		IF NOT Busy 
		THEN (* Busy initalisation is TRUE *)
			Busy := BusyIntern 								:= TRUE;
			state 											:= eSTATE.ABORTING;
		ELSE
			; (* Wait for Startup End*)
		END_IF
	{endregion} 		
	{region "IDLE"} 
	eSTATE.IDLE:
		info 												:= TO_STRING(eSTATE.IDLE);
		
		IF GoToAborting 
		THEN
			Busy := BusyIntern 								:= TRUE; 
			state 											:= eSTATE.ABORTING;
		ELSIF RemoteCtrlEnable AND MasterCmdState = eSTATE.STOPPING 
		THEN
			Busy := BusyIntern 								:= TRUE; 
			state 											:= eSTATE.STOPPING;
		ELSIF NOT RemoteCtrlEnable AND SetMode <> eMODE.IDLE
			OR 
			RemoteCtrlEnable
			AND MasterCmdState <> eSTATE.IDLE
			AND MasterCmdState <> eSTATE.RESETTING
		THEN
			Busy := BusyIntern 								:= TRUE; 
			Mode 											:= SEL(RemoteCtrlEnable,SetMode,MasterCmdMode);
			State 											:= eSTATE.STARTING;
		ELSE
			Mode 											:= eMODE.IDLE;
		END_IF
	{endregion} 
	{region "STARTING"} 	
	eSTATE.STARTING: info 									:= TO_STRING(eSTATE.STARTING);
	
		IF GoToAborting 
		THEN
			state 											:= eSTATE.ABORTING;
			Busy := BusyIntern 								:= TRUE;

		ELSIF RemoteCtrlEnable
			AND(
			MasterCmdState = eSTATE.STOPPING
			OR (* Betriebsartenwechsel ueber RemoteCtrl ein *)
			NOT RemoteDataToSlaves._WORDS[2].8 AND Mode <> MasterCmdMode)
		THEN
			state 											:= eSTATE.STOPPING;
			Busy := BusyIntern 								:= TRUE;
		ELSIF NOT Busy 
		THEN
			state 											:= eSTATE.STARTED;			
		END_IF
	{endregion} 		
	{region "STARTED"} 	
	eSTATE.STARTED: info 									:= TO_STRING(eSTATE.STARTED);
		
		IF GoToAborting 
		THEN
			Busy := BusyIntern 								:= TRUE; 
			state 											:= eSTATE.ABORTING;
		ELSIF RemoteCtrlEnable
			AND NOT RemoteDataToSlaves._WORDS[2].8 
			AND Mode <> MasterCmdMode
		THEN (* Betriebsartenwechsel ueber RemoteCtrl ein *)
			Busy := BusyIntern 								:= TRUE; 
			state 											:= eSTATE.STOPPING;
		ELSIF NOT RemoteCtrlEnable
			OR 	
			RemoteCtrlEnable
			AND MasterCmdState <> eSTATE.STARTED
			AND MasterCmdState <> eSTATE.STARTING
		THEN
			IF RemoteCtrlEnable AND MasterCmdState = eSTATE.EXECUTE
				OR NOT RemoteCtrlEnable
			THEN
				Busy := BusyIntern 							:= TRUE; 
				state 										:= eSTATE.EXECUTE;
			ELSIF RemoteCtrlEnable AND Options.5 //Compl. aktiviert
				AND(MasterCmdState = eSTATE.COMPLETING OR	MasterCmdState = eSTATE.COMPLETE)
			THEN
				Busy := BusyIntern 							:= TRUE; 
				state 										:= eSTATE.COMPLETING;
			ELSE
				Busy := BusyIntern 							:= TRUE; 
				state 										:= eSTATE.STOPPING;
			END_IF
		END_IF
	{endregion} 	
	{region "EXECUTE"} 
	eSTATE.EXECUTE: info 									:= TO_STRING(eSTATE.EXECUTE);
	
		IF GoToAborting 
		THEN
			Busy := BusyIntern 								:= TRUE; 
			state 											:= eSTATE.ABORTING;

		ELSIF SetMode <> Mode
			AND NOT RemoteCtrlEnable
			AND NOT Options.1  (* Modewechsel ueber Stopping/Completing wenn Options.1 nicht gesetzt *)
			OR	
			NOT RemoteCtrlEnable
			AND SetMode = eMODE.IDLE
			OR	
			RemoteCtrlEnable
			AND MasterCmdState <> eSTATE.EXECUTE
			AND MasterCmdState <> eSTATE.STARTING
			AND MasterCmdState <> eSTATE.STARTED
			OR (* Betriebsartenwechsel ueber RemoteCtrl ein *)
			RemoteCtrlEnable
			AND NOT RemoteDataToSlaves._WORDS[2].8 AND Mode <> MasterCmdMode
		THEN
			IF Options.5 (* Mode change over Completing *)
				AND(MasterCmdState = eSTATE.COMPLETING
				AND RemoteCtrlEnable
				OR	
				NOT RemoteCtrlEnable)
			THEN
				Busy := BusyIntern 							:= TRUE; 
				state 										:= eSTATE.COMPLETING;
			ELSE      						
				Busy := BusyIntern 							:= TRUE; 				
				state 										:= eSTATE.STOPPING;
			END_IF

		ELSIF Options.1  (* Modewechsel in Execute *)
			AND(
			SetMode <> Mode AND NOT RemoteCtrlEnable
			OR	
			MasterCmdMode <> Mode AND RemoteCtrlEnable)
		THEN
			Mode 											:= SEL(RemoteCtrlEnable,SetMode,MasterCmdMode);

		ELSIF RemoteCtrlEnable
			AND(
			MasterCmdState = eSTATE.HOLDING 
			OR MasterCmdState = eSTATE.HELD) 
		THEN
			Busy := BusyIntern 								:= TRUE; 
			state 											:= eSTATE.HOLDING;
		ELSIF RemoteCtrlEnable
			AND(
			MasterCmdState = eSTATE.SUSPENDING 
			OR MasterCmdState = eSTATE.SUSPENDED) 
		THEN
			Busy := BusyIntern 								:= TRUE; 
			state 											:= eSTATE.SUSPENDING;
		END_IF
	{endregion} 	
	{region "SUSPENDING"} 
	eSTATE.SUSPENDING: 	info 								:= TO_STRING(eSTATE.SUSPENDING);	
		
		IF GoToAborting 
		THEN
			state 											:= eSTATE.ABORTING;
			Busy := BusyIntern 								:= TRUE;

		ELSIF RemoteCtrlEnable
			AND(
			MasterCmdState = eSTATE.STOPPING
			OR (* Betriebsartenwechsel ueber RemoteCtrl ein *)
			NOT RemoteDataToSlaves._WORDS[2].8 AND Mode <> MasterCmdMode)
		THEN
			state 											:= eSTATE.STOPPING;
			Busy := BusyIntern 								:= TRUE;
		ELSIF NOT Busy 
		THEN
			state 											:= eSTATE.SUSPENDED;		
		END_IF	
	{endregion} 	
	{region "SUSPENDED"} 
	eSTATE.SUSPENDED:	info 								:= TO_STRING(eSTATE.SUSPENDED);	
	
		IF GoToAborting 
		THEN
			Busy := BusyIntern 								:= TRUE; 
			state 											:= eSTATE.ABORTING;
		ELSIF RemoteCtrlEnable
			AND NOT RemoteDataToSlaves._WORDS[2].8 
			AND Mode <> MasterCmdMode
		THEN (* Betriebsartenwechsel ueber RemoteCtrl ein *)
			Busy := BusyIntern 								:= TRUE; 
			state 											:= eSTATE.STOPPING;
		ELSIF NOT RemoteCtrlEnable
			OR 	
			RemoteCtrlEnable
			AND MasterCmdState <> eSTATE.SUSPENDED
			AND MasterCmdState <> eSTATE.SUSPENDING
		THEN
			IF RemoteCtrlEnable 
				AND(MasterCmdState = eSTATE.UNSUSPENDING OR MasterCmdState = eSTATE.EXECUTE OR MasterCmdState = eSTATE.COMPLETING)
				OR NOT RemoteCtrlEnable
			THEN
				Busy := BusyIntern 							:= TRUE; 
				state 										:= eSTATE.UNSUSPENDING;	
			ELSE
				Busy := BusyIntern 							:= TRUE; 
				state 										:= eSTATE.STOPPING;
			END_IF
		END_IF
	{endregion} 	
	{region "UNSUSPENDING"}	
	eSTATE.UNSUSPENDING: info 								:= TO_STRING(eSTATE.UNSUSPENDING);
	
		IF GoToAborting 
		THEN
			state 											:= eSTATE.ABORTING;
			Busy := BusyIntern 								:= TRUE;

		ELSIF RemoteCtrlEnable
			AND(
			MasterCmdState = eSTATE.STOPPING
			OR (* Betriebsartenwechsel ueber RemoteCtrl ein *)
			NOT RemoteDataToSlaves._WORDS[2].8 AND Mode <> MasterCmdMode)
		THEN
			state 											:= eSTATE.STOPPING;
			Busy := BusyIntern 								:= TRUE;
		ELSIF NOT Busy 
		THEN
			Busy := BusyIntern 								:= TRUE; 
			state											:= eSTATE.EXECUTE;
		END_IF
	{endregion} 	
	{region "HOLDING"}	
	eSTATE.HOLDING:		info 								:= TO_STRING(eSTATE.HOLDING);
	
		IF GoToAborting 
		THEN
			state 											:= eSTATE.ABORTING;
			Busy := BusyIntern 								:= TRUE;

		ELSIF RemoteCtrlEnable
			AND(
			MasterCmdState = eSTATE.STOPPING
			OR (* Betriebsartenwechsel ueber RemoteCtrl ein *)
			NOT RemoteDataToSlaves._WORDS[2].8 AND Mode <> MasterCmdMode)
		THEN
			state 											:= eSTATE.STOPPING;
			Busy := BusyIntern 								:= TRUE;
		ELSIF NOT Busy 
		THEN
			state 											:= eSTATE.HELD;		
		END_IF	
	{endregion} 	
	{region "HELD"}	
	eSTATE.HELD:		info 								:= TO_STRING(eSTATE.HELD);
	
		IF GoToAborting 
		THEN
			Busy := BusyIntern 								:= TRUE; 
			state 											:= eSTATE.ABORTING;
		ELSIF RemoteCtrlEnable
			AND NOT RemoteDataToSlaves._WORDS[2].8 
			AND Mode <> MasterCmdMode
		THEN (* Betriebsartenwechsel ueber RemoteCtrl ein *)
			Busy := BusyIntern 								:= TRUE; 
			state 											:= eSTATE.STOPPING;
		ELSIF NOT RemoteCtrlEnable
			OR 	
			RemoteCtrlEnable
			AND MasterCmdState <> eSTATE.HELD
			AND MasterCmdState <> eSTATE.HOLDING
		THEN
			IF RemoteCtrlEnable 
				AND(MasterCmdState = eSTATE.EXECUTE OR MasterCmdState = eSTATE.UNHOLDING OR MasterCmdState = eSTATE.COMPLETING)
				OR NOT RemoteCtrlEnable
			THEN
				Busy := BusyIntern 							:= TRUE; 
				state 										:= eSTATE.UNHOLDING;	
			ELSE
				Busy := BusyIntern 							:= TRUE; 
				state 										:= eSTATE.STOPPING;
			END_IF
		END_IF
	{endregion} 	
	{region "UNHOLDING"}	
	eSTATE.UNHOLDING: 	info 								:= TO_STRING(eSTATE.UNHOLDING);
	
		IF GoToAborting 
		THEN
			state 											:= eSTATE.ABORTING;
			Busy := BusyIntern 								:= TRUE;

		ELSIF RemoteCtrlEnable
			AND(
			MasterCmdState = eSTATE.STOPPING
			OR (* Betriebsartenwechsel ueber RemoteCtrl ein *)
			NOT RemoteDataToSlaves._WORDS[2].8 AND Mode <> MasterCmdMode)
		THEN
			state 											:= eSTATE.STOPPING;
			Busy := BusyIntern 								:= TRUE;
		ELSIF NOT Busy 
		THEN
			Busy := BusyIntern 								:= TRUE; 
			state											:= eSTATE.EXECUTE;
		END_IF
	{endregion} 	
	{region "COMPLETING"}	
	eSTATE.COMPLETING: info 								:= TO_STRING(eSTATE.COMPLETING);
	
		IF GoToAborting 
		THEN
			Busy := BusyIntern 								:= TRUE; 
			state 											:= eSTATE.ABORTING;

		ELSIF RemoteCtrlEnable
			AND( (* Betriebsartenwechsel ueber RemoteCtrl ein *)
			MasterCmdState = eSTATE.STOPPING
			OR 
			NOT RemoteDataToSlaves._WORDS[2].8  AND Mode <> MasterCmdMode)
			OR	
			NOT RemoteCtrlEnable AND NOT Options.5 (* Cancel Completing *)
		THEN
			Busy := BusyIntern 								:= TRUE; 
			state 											:= eSTATE.STOPPING;

		ELSIF NOT Busy
		THEN
			state 											:= eSTATE.COMPLETE;
		END_IF
	{endregion} 	
	{region "COMPLETE"}	
	eSTATE.COMPLETE: info 									:= TO_STRING(eSTATE.COMPLETE);
		
		IF GoToAborting 
		THEN
			Busy := BusyIntern 								:= TRUE; 
			state 											:= eSTATE.ABORTING;

		ELSIF NOT RemoteCtrlEnable
			OR	
			RemoteCtrlEnable
			AND MasterCmdState <> eSTATE.COMPLETE
			AND MasterCmdState <> eSTATE.COMPLETING
		THEN
			Busy := BusyIntern 								:= TRUE; 
			state 											:= eSTATE.STOPPING;
		END_IF
	{endregion} 	
	{region "ABORTING"}	
	eSTATE.ABORTING: info 									:= TO_STRING(eSTATE.ABORTING);
		IF NOT Busy
			OR NOT EStopDelayOK
			OR RemoteCtrlEnable AND NOT MasterCmdInfo.15 (* EStop Delay False *)
		THEN
			StateComplete(); (* Ueber Hardware vorgegeben *)
			state 											:= eSTATE.ABORTED;
		END_IF
			 
		(* Set SubCtrl Busy if state changing *)
		IF state <> eSTATE.ABORTING AND state <> eSTATE.ABORTED 
		THEN 
			Busy := BusyIntern 								:= TRUE; 
		END_IF
			 
	{endregion} 	
	{region "ABORTED"}	
	eSTATE.ABORTED: info 									:= TO_STRING(eSTATE.ABORTED);
		
		IF NOT RemoteCtrlEnable AND EStopDirectOK AND EStopDelayOK
			OR 	
			RemoteCtrlEnable
			AND(EStopDirectOK AND EStopDelayOK OR Options.3)
			AND MasterCmdState <> eSTATE.ABORTED
			AND MasterCmdState <> eSTATE.ABORTING
			AND MasterCmdState <> eSTATE.STARTUP
		THEN
			Busy := BusyIntern 								:= TRUE; 
			state 											:= eSTATE.CLEARING;
		ELSE			
			(* Ack error in aborted *)
			IF LocalReset
			THEN
		 		ErrHdl.reset();
			END_IF
		END_IF
		
		(* set Mode *)
		IF Options.0
		THEN
			Mode 											:= eMODE.IDLE;
		ELSE (* take the current mode back *)
			Mode 											:= SEL(RemoteCtrlEnable,SetMode,MasterCmdMode);
		END_IF
	{endregion} 	
	{region "CLEARING"}	
	eSTATE.CLEARING: info 									:= TO_STRING(eSTATE.CLEARING);
		
		IF GoToAborting 
		THEN
			Busy := BusyIntern 								:= TRUE; 
			state 											:= eSTATE.ABORTING;
		ELSIF NOT Busy
			AND(EStopOK OR Options.3) (* Local EStop Disabled *)
			AND(MasterCmdInfo.14 OR NOT RemoteCtrlEnable) (* RemoteCtrl EStop OK *)
		THEN
			state 											:= eSTATE.STOPPED;
		END_IF
	{endregion} 	
	{region "STOPPING"}	
	eSTATE.STOPPING: Info									:= TO_STRING(eSTATE.STOPPING);
		
		IF GoToAborting 
		THEN
			Busy := BusyIntern 								:= TRUE; 
			state 											:= eSTATE.ABORTING;
		ELSIF NOT Busy 
		THEN
			state 											:= eSTATE.STOPPED;
		END_IF
	{endregion} 	
	{region "STOPPED"}	
	eSTATE.STOPPED: info 									:= TO_STRING(eSTATE.STOPPED);
		
		IF GoToAborting 
		THEN
			Busy := BusyIntern 								:= TRUE; 
			state 											:= eSTATE.ABORTING;
		ELSIF LocalReset AND ErrHdl.flag
			AND(NOT RemoteCtrlEnable OR MasterCmdState <> eSTATE.STOPPED) (* Weiter ueber Quitt im Fehlerfall *)
			AND(ErrHdl.id <> ERROR_MACHINE OR NOT Options.4)
			OR 
			NOT RemoteCtrlEnable
			AND(NOT ErrHdl.flag OR NOT Options.6 AND ErrHdl.id <> ERROR_EXTERNAL) (* Automatisch weiter wenn kein Fehler, oder ACK nicht erforderlich und Fehler nicht Extern (Quittierung erfolgt dort)*)
			OR	
			RemoteCtrlEnable (* Weiter wenn Remote Unit nicht in Stopped/Completing und nicht in Fehler *)
			AND MasterCmdState <> eSTATE.STOPPED
			AND MasterCmdState <> eSTATE.STOPPING
			AND MasterCmdState <> eSTATE.CLEARING
			AND MasterCmdState <> eSTATE.COMPLETING 
			AND MasterCmdState <> eSTATE.COMPLETE
			AND(NOT ErrHdl.flag OR NOT Options.6)
			OR 
			RemoteCtrlEnable (* Weiter wenn Maschinenfehler resetet wird *)
			AND MasterCmdState = eSTATE.RESETTING
			AND ErrHdl.flag //(MasterCmdInfo.11 or MasterCmdInfo.12 OR MasterCmdInfo.13) //OR ErrHdl.id = ERROR_MACHINE ist Bit 12)
		THEN
			Busy := BusyIntern 								:= TRUE; 
			ErrHdl.reset();
			state 											:= eSTATE.RESETTING;
		END_IF
	
		(* set Mode *)
		IF Options.0 
		THEN
			Mode 											:= eMODE.IDLE;
		ELSE (* take the current mode back *)
			Mode 											:= SEL(RemoteCtrlEnable,SetMode,MasterCmdMode);
		END_IF
	{endregion} 	
	{region "RESETTING"}	
	eSTATE.RESETTING: info 									:= TO_STRING(eSTATE.RESETTING);
		
		IF GoToAborting 
		THEN
			Busy := BusyIntern 								:= TRUE; 
			state 											:= eSTATE.ABORTING;
		ELSIF MasterCmdState = eSTATE.STOPPING 
			AND RemoteCtrlEnable 
		THEN
			Busy := BusyIntern 								:= TRUE; 
			state 											:= eSTATE.STOPPING;
		ELSIF NOT Busy 
		THEN
			state 											:= eSTATE.IDLE;
		END_IF
	{endregion} 	

	ELSE
		info 												:= CONCAT('ERROR unkown state ', TO_STRING(state));
		ErrHdl.flag 										:= TRUE;
		ErrHdl.fnc 											:= 'SubCtrl';
		ErrHdl.id											:= 99;
		ErrHdl.state										:= state;
		ErrHdl.text 										:= CONCAT('unkown state:',DINT_TO_STRING(ErrHdl.state));
		SetLocalError();
	END_CASE
		 
(* State Check *************************************************)
	RT_StateChanged 										:= LastState <> State;
	LastState 												:= State;
	
(* Statebits ***********************************************************************************)
	InStartup												:= state = eSTATE.STARTUP;
	InIdle													:= state = eSTATE.IDLE;
	InStarting												:= state = eSTATE.STARTING;
	InStarted												:= state = eSTATE.STARTED;
	InExecute												:= state = eSTATE.EXECUTE;
	InCompleting											:= state = eSTATE.COMPLETING;
	InComplete												:= state = eSTATE.COMPLETE;
	InAborting												:= state = eSTATE.ABORTING;
	InAborted												:= state = eSTATE.ABORTED;
	InClearing												:= state = eSTATE.CLEARING;
	InStopping												:= state = eSTATE.STOPPING;
	InStopped												:= state = eSTATE.STOPPED;
	InResetting												:= state = eSTATE.RESETTING;

	EStopStartupOK											:= 	NOT InAborted 
																AND(
																EStopStartupOK 
																OR 
																NOT InAborting AND NOT InClearing 
																AND NOT InStartup AND NOT InStopped );
                    										
(* optional
	InSuspending	:= state = eSTATE.SUSPENDING;
	InSuspended		:= state = eSTATE.SUSPENDED;
	InUnsuspending	:= state = eSTATE.UNSUSPENDING;

	InHolding		:= state = eSTATE.HOLDING;
	InHeld			:= state = eSTATE.HELD;
	InUnholding		:= state = eSTATE.UNHOLDING;
*)

(***************************************************************)
(* Read Subs Status and synchronize							   *)
(***************************************************************)		
{region "Check slave states and send command"}	
	(* Init Flag, all Subs in same state *)
	NoSlavesConnected										:= TRUE;
	SlavesInSync 											:= NOT RT_StateChanged;
	SlavesBusy    											:= FALSE;
	NoOfBusySlaves											:= 0;
	(* Init remote command data to slaves  *)
	RemoteDataToSlaves._INTs[0]								:= Mode;
	RemoteDataToSlaves._WORDS[2]							:= TO_WORD(Options);
	RemoteDataToSlaves._WORDS[2].8							:= RemoteCtrlEnable;
	RemoteDataToSlaves._WORDS[2].9							:= LocalReset;	
	RemoteDataToSlaves._WORDS[2].14							:= EStopOK OR Options.3;
	RemoteDataToSlaves._WORDS[2].15							:= EStopDelayOK OR Options.3;	
	RemoteDataToSlaves._INTs[3]								:= Id;
		
	(* read Subs state an send cmd to all subs *)
	FOR i := MIN_SLAVE TO MAX_SLAVE DO
		IF ipSlave[i] <> 0 
		THEN 
			NoSlavesConnected 								:= FALSE;(* pointer is used *)
			RemoteDataFromSlave								:= ipSlave[i].remoteData; //Read remote status data from slaves
			IF RemoteDataFromSlave._WORDS[2].8 
			THEN (* External Sub is Remote-Controlled *)
				(* Check the status from then external subs *)
				IF((RemoteDataFromSlave._WORDS[2].11 OR RemoteDataFromSlave._WORDS[2].13) 
					AND RemoteDataFromSlave._WORDS[2].4)(* Maschine to Remotesystem if Enabled, or External Error *)
					AND NOT ErrHdl.flag
					AND NOT InStartup AND NOT InResetting
					AND NOT InAborting AND NOT InAborted
				THEN (* external sub has fatal error *)
					(* external subs send fatal machine error -> bring local sub in Stopping with error *)
					ErrHdl.flag								:= TRUE;
					ErrHdl.state							:= state;
					ErrHdl.fnc 								:= name;
					ErrHdl.id								:= ERROR_EXTERNAL;
					ErrHdl.text 							:= CONCAT('Fatal machine error in Sub index no.:',INT_TO_STRING(i));
					Busy									:= state <> eSTATE.STOPPING;
					state 									:= eSTATE.STOPPING;
					SlavesInSync 							:= FALSE;
				ELSE (* external sub has no error *)
					IF SlavesState = RemoteDataFromSlave._INTs[1]
					THEN (* Check if sub is in sync with other subs *)
						SlavesState 						:= RemoteDataFromSlave._INTs[1];
					ELSE (* external sub is not in sync with other subs *)
						IF (RemoteDataFromSlave._INTs[1] = eSTATE.ABORTED OR RemoteDataFromSlave._INTs[1] = eSTATE.ABORTING)
							AND NOT InAborted 
							AND NOT InAborting
							AND NOT RemoteDataFromSlave._WORDS[2].3 (* Local EStop-Signals Disable *)
							OR RemoteDataFromSlave._WORDS[2].11 (* Maschine Error *)
							OR RemoteDataFromSlave._WORDS[2].12 (* Local Error  *)
							OR RemoteDataFromSlave._WORDS[2].13 (* External Error  *)
							OR (* comleting at sub disabled *)
							NOT RemoteDataFromSlave._WORDS[2].5 
							AND(InCompleting OR InComplete)
							AND(RemoteDataFromSlave._INTs[1] = eSTATE.STOPPING OR RemoteDataFromSlave._INTs[1] = eSTATE.STOPPED)
						THEN
							; (* ignore cause sub use local EStop-signals, or error in stopped *)
						ELSE
							SlavesState						:= RemoteDataFromSlave._INTs[1];
							SlavesInSync 					:= FALSE;
						END_IF
					END_IF

					(* subs busy *)
					IF (RemoteDataFromSlave._INTs[1] = eSTATE.ABORTED OR RemoteDataFromSlave._INTs[1] = eSTATE.ABORTING )
						AND NOT InAborted 
						AND NOT InAborting
						AND NOT RemoteDataFromSlave._WORDS[2].3 (* Local EStop-Signals Disable *)
						OR RemoteDataFromSlave._WORDS[2].12 (* Local Error *)
						OR 
						SlavesState = eSTATE.EXECUTE AND NOT InExecute
					THEN
						; (* ignore cause sub is in error or use local EStop-Signals *)
					ELSIF RemoteDataFromSlave._WORDS[2].10 
					THEN
						SlavesBusy 							:= TRUE;
						NoOfBusySlaves						:= NoOfBusySlaves + 1;
					END_IF

				END_IF
			ELSE (* external Sub is not in RemoteCtrl *)
				;
			END_IF

			(* Write latest command data   *)
			RemoteDataToSlaves._INTs[1]						:= State;
			RemoteDataToSlaves._WORDS[2].10					:= Busy;
			RemoteDataToSlaves._WORDS[2].11					:= ErrHdl.id = ERROR_MACHINE;
			RemoteDataToSlaves._WORDS[2].12					:= ErrHdl.id = ERROR_LOCAL;
			RemoteDataToSlaves._WORDS[2].13					:= ErrHdl.id = ERROR_EXTERNAL;

			(* set slave command data *)
			ipSlave[i].remoteData							:= RemoteDataToSlaves; //Write data as command to every slave
		ELSE
			EXIT; (* pointer not used -> Exit for *)
		END_IF
	END_FOR

	(* Set state complete only if all Subs in the same state or current state is Execute *)
	IF SlavesInSync AND NOT NoSlavesConnected 
	THEN //Subs in sync
		IF SlavesBusy 
			OR (BusyIntern AND Options.2) 
			OR (NOT EStopOK AND NOT Options.3 AND InClearing) (* Solange Busy halten, biss durch EStopOK aus Clearing gegangen werden kann *)
		THEN
			; (* al least one sub is busy or not StateComplete *)
		ELSIF Busy 
		THEN
			Busy := BusyIntern 								:= FALSE; (* All subs not StateComplete (NOT Busy) set UnitSub StateComplete *)
		END_IF
	END_IF
{endregion}
	 
(* Set Status RemoteData for master to check ************************************************************)
	RemoteDataToSlaves._INTs[0] 							:= Mode;
	RemoteDataToSlaves._INTs[1]								:= State;
	RemoteDataToSlaves._WORDs[2]							:= TO_WORD(Options);
	RemoteDataToSlaves._WORDs[2].8							:= RemoteCtrlEnable;
	RemoteDataToSlaves._WORDs[2].9							:= LocalReset;
	RemoteDataToSlaves._WORDs[2].10							:= Busy;
	RemoteDataToSlaves._WORDs[2].11							:= ErrHdl.id = ERROR_MACHINE;
	RemoteDataToSlaves._WORDs[2].12							:= ErrHdl.id = ERROR_LOCAL;
	RemoteDataToSlaves._WORDs[2].13							:= ErrHdl.id = ERROR_EXTERNAL;
	RemoteDataToSlaves._WORDs[2].14							:= EStopOK OR Options.3;
	RemoteDataToSlaves._WORDs[2].15							:= EStopDelayOK OR Options.3;
	RemoteDataToSlaves._INTs[3]								:= Id;
	

(* Reset LocalAck ******************************************************************************)
	Localreset												:= FALSE;

(***********************************************************************************************)

METHOD PRIVATE FINAL _createID : INT
VAR_STAT //Value is stored for each instance
	IdCnt													: INT;
END_VAR
IdCnt														:= IdCnt + 1;
_CreateID 													:= IdCnt;
END_METHOD

METHOD PUBLIC FINAL addSlave : BOOL
VAR_INPUT
	ipSlave													:	I_Statemodel;
END_VAR
addSlave													:= FALSE;	
IF ipSlave <> 0	
then
	FOR i := MIN_SLAVE TO MAX_SLAVE
	DO 
		IF ipSlave = THIS^.ipSlave[i] THEN
			addSlave										:= TRUE;
			EXIT;
		ELSIF THIS^.ipSlave[i] = 0
		THEN								
			THIS^.ipSlave[i]								:= ipSlave;
			addSlave										:= TRUE;
			EXIT;
		END_IF
	END_FOR
END_IF
END_METHOD

METHOD FB_init : BOOL
VAR_INPUT
	bInitRetains : BOOL; // if TRUE, the retain variables are initialized (warm start / cold start)
	bInCopyCode : BOOL;  // if TRUE, the instance afterwards gets moved into the copy code (online change)
END_VAR
(* Generate ID ****************************************************)
	IF Id = 0 
	THEN 
		id 													:= _CreateID(); 
		IF Name = '' 
		THEN 
			Name 											:= CONCAT('Statemodel Id ',TO_STRING(Id)); 
		ELSE
			Name 											:= CONCAT(Name , CONCAT(' Id ', TO_STRING(Id))); 
		END_IF
	END_IF	
(***********************************************************************)
END_METHOD

METHOD PUBLIC goToStopping : BOOL //TRUE = stopping activated
VAR_INPUT
END_VAR

CASE State OF
eSTATE.IDLE,
eSTATE.STARTING,
eSTATE.STARTED,	
eSTATE.EXECUTE,
eSTATE.SUSPENDING,
eSTATE.SUSPENDED,
eSTATE.UNSUSPENDING,	
eSTATE.HOLDING,
eSTATE.HELD,
eSTATE.UNHOLDING,	
eSTATE.COMPLETING,
eSTATE.COMPLETE,
eSTATE.STOPPING,
eSTATE.STOPPED,
eSTATE.RESETTING:
	state 													:= eSTATE.STOPPING;
	Busy := BusyIntern 										:= TRUE;
	goToStopping											:= TRUE;
ELSE
(*	
	eSTATE.STARTUP,
	eSTATE.ABORTING,
	eSTATE.ABORTED,
	eSTATE.CLEARING:
*)	
	goToStopping											:= FALSE;
END_CASE
END_METHOD

METHOD PUBLIC isModeActive : BOOL
VAR_INPUT
	Mode													: eMODE;				
END_VAR
IsModeActive := Mode = THIS^.Mode AND(InExecute OR InCompleting);
END_METHOD

METHOD PUBLIC isStateActive : BOOL
VAR_INPUT
	state								: eSTATE;
END_VAR
IsStateActive := state = This^.State;
END_METHOD

METHOD PUBLIC reset : boOL //Result = TRUE if Resetting finished - ErrHdl.Flag = FALSE
VAR_INPUT
END_VAR
LocalReset													:= TRUE;
reset														:= NOT ErrHdl.flag;
END_METHOD

METHOD PUBLIC setLocalError : booL
VAR_INPUT
END_VAR
IF NOT ErrHdl.flag
	AND state <> eSTATE.ABORTING
	AND state <> eSTATE.ABORTED
	AND state <> eSTATE.CLEARING
	and state <> eSTATE.RESETTING
THEN
	ErrHdl.flag 											:= TRUE;
	ErrHdl.state											:= state;
	ErrHdl.fnc												:= name;
	ErrHdl.id												:= ERROR_LOCAL;
	ErrHdl.text 											:= 'Local ctrl error';
	Busy													:= state <> eSTATE.STOPPING;
	state 													:= eSTATE.STOPPING;
	SetLocalError											:= TRUE;
ELSE
	SetLocalError											:= ErrHdl.id = ERROR_LOCAL;
END_IF
END_METHOD

METHOD PUBLIC setMachineError : booL
VAR_INPUT
END_VAR
IF NOT ErrHdl.flag
	AND state <> eSTATE.ABORTING
	AND state <> eSTATE.ABORTED
	AND state <> eSTATE.CLEARING
	AND state <> eSTATE.RESETTING
THEN
	ErrHdl.flag												:= TRUE;
	ErrHdl.state											:= state;
	ErrHdl.fnc												:= name;
	ErrHdl.id												:= ERROR_MACHINE;
	ErrHdl.text 											:= 'Fatal machine error';
	Busy													:= state <> eSTATE.STOPPING;
	state 													:= eSTATE.STOPPING;
	SetMachineError											:= TRUE;
ELSE
	SetMachineError											:= ErrHdl.id = ERROR_MACHINE;;
END_IF
END_METHOD

METHOD PUBLIC FINAL stateComplete : BOOL //Result = TRUE if state completed (BusyIntern=FALSE)
VAR_INPUT
END_VAR
BusyIntern 													:= FALSE;
StateComplete												:= NOT BusyIntern AND NOT Busy;
END_METHOD

{attribute 'monitoring' := 'call'}
PROPERTY PUBLIC optDisableSafetyInputs : BOOL
GET
optDisableSafetyInputs := Options.3;
END_GET
SET
Options.3 := optDisableSafetyInputs;
END_SET
END_PROPERTY

{attribute 'monitoring' := 'call'}
PROPERTY PUBLIC optEnableAutoChangeModeToIdle : BOOL
GET
optEnableAutoChangeModeToIdle := Options.0;
END_GET
SET
Options.0 := optEnableAutoChangeModeToIdle;
END_SET
END_PROPERTY

{attribute 'monitoring' := 'call'}
PROPERTY PUBLIC optEnableExplicitReset : BOOL
GET
optEnableExplicitReset := Options.6;
END_GET
SET
Options.6 := optEnableExplicitReset;
END_SET
END_PROPERTY

{attribute 'monitoring' := 'call'}
PROPERTY PUBLIC optEnableExternalStateComplete : BOOL
GET
optEnableExternalStateComplete := Options.2;
END_GET
SET
Options.2 := optEnableExternalStateComplete;
END_SET
END_PROPERTY

{attribute 'monitoring' := 'call'}
PROPERTY PUBLIC optEnableFwdMachineErrorToMaster : BOOL
GET
optEnableFwdMachineErrorToMaster := Options.4;
END_GET
SET
Options.4 := optEnableFwdMachineErrorToMaster;
END_SET
END_PROPERTY

{attribute 'monitoring' := 'call'}
PROPERTY PUBLIC optEnableModeChangeInExecute : BOOL
GET
optEnableModeChangeInExecute := Options.1;
END_GET
SET
Options.1 := optEnableModeChangeInExecute;
END_SET
END_PROPERTY

{attribute 'monitoring' := 'call'}
PROPERTY PUBLIC optEnableModeChangeViaStateCompl : BOOL
GET
optEnableModeChangeViaStateCompl := Options.5;
END_GET
SET
Options.5 := optEnableModeChangeViaStateCompl;
END_SET
END_PROPERTY

{attribute 'monitoring' := 'call'}
PROPERTY PUBLIC optEnableSetActState : BOOL
GET
optEnableSetActState := Options.7;
END_GET
SET
Options.7 := optEnableSetActState;
END_SET
END_PROPERTY

{attribute 'monitoring' := 'call'}
PROPERTY public actMode : eMODE
GET
actMode := Mode;
END_GET
END_PROPERTY

{attribute 'monitoring' := 'call'}
//Actual state enum, only read access by default, check options for further information 
PROPERTY public actState : eSTATE
GET
actState := state;
END_GET
SET
PUBLIC //Use with care!! 
VAR
END_VAR
IF Options.7  //OPTION_ENABLE_SET_ACT_STATE
THEN
	IF actState <> State
	THEN
		state 													:= actState;
		Busy := BusyIntern 										:= TRUE;	
	END_IF
ELSE	
	ErrHdl.flag 												:= TRUE;
	ErrHdl.state												:= state;
	ErrHdl.fnc													:= name;
	ErrHdl.id													:= ERROR_LOCAL;
	ErrHdl.text 												:= 'Write "actState" not allowed, use OPTION_ENABLE_SET_ACT_STATE to enable set actState';
	Busy														:= state <> eSTATE.STOPPING;
	state 														:= eSTATE.STOPPING;
END_IF
END_SET
END_PROPERTY

{attribute 'monitoring' := 'call'}
PROPERTY PUBLIC ipMasterUnit : I_Statemodel //The slave will add his interface pointer into the master through this propertiy
SET
IF IdRemoteMaster = 0 AND_THEN ipMasterUnit <> 0
THEN
	RemoteDataToSlaves									:= ipMasterUnit.remoteData;	
	IF IdRemoteMaster <> RemoteDataToSlaves._INTs[3] 
	THEN
		IF ipMasterUnit.addSlave(THIS^)
		THEN					
			remoteData 									:= RemoteDataToSlaves; 
		END_IF
	END_IF
END_IF
END_SET
END_PROPERTY

{attribute 'monitoring' := 'call'}
PROPERTY isBusy : BOOL
GET
isBusy := Busy;
END_GET
END_PROPERTY

PROPERTY public remoteData : U_64BIT_DATATYPE
GET
//statis of sub
remoteData := RemoteDataToSlaves;
END_GET
SET
//Cmd to sub
MasterCmdMode 	:= remoteData._INTs[0];
MasterCmdState := remoteData._INTs[1];
MasterCmdInfo 	:= remoteData._WORDS[2];
IdRemoteMaster := remoteData._INts[3];
END_SET
END_PROPERTY

{attribute 'monitoring' := 'call'}
PROPERTY PUBLIC rErrHdl : REFERENCE to ERROR_HDL
GET
rErrHdl REF= Errhdl;
END_GET
END_PROPERTY

PROPERTY PUBLIC setStateComplete : BOOL
GET
SetStateComplete := not BusyIntern and not Busy;
END_GET
SET
IF SetStateComplete AND BusyIntern
THEN
	StateComplete();
END_IF
END_SET
END_PROPERTY

END_FUNCTION_BLOCK

// POUs/Statemodel/control/I_Statemodel
INTERFACE I_Statemodel extends I_StatemodelBase

METHOD PUBLIC FINAL addSlave : BOOL
VAR_INPUT
	ipSlave					:	I_Statemodel;
END_VAR
END_METHOD

METHOD PUBLIC isModeActive : BOOL
VAR_INPUT
	Mode													: eMODE;				
END_VAR
END_METHOD

METHOD PUBLIC isStateActive : BOOL
VAR_INPUT
	state						:	eSTATE;
END_VAR
END_METHOD

METHOD PUBLIC reset : boOL //Result = TRUE if Resetting finished - ErrHdl.Flag = FALSE
VAR_INPUT
END_VAR
END_METHOD

METHOD PUBLIC setLocalError : booL
VAR_INPUT
END_VAR
END_METHOD

PROPERTY public remoteData : U_64BIT_DATATYPE
GET
END_GET
SET
END_SET
END_PROPERTY

{attribute 'monitoring' := 'call'}
PROPERTY PUBLIC rErrHdl : REFERENCE to ERROR_HDL
GET
END_GET
END_PROPERTY

END_INTERFACE

// POUs/Statemodel/control/I_StatemodelBase
INTERFACE I_StatemodelBase Extends __System.IQueryInterface

METHOD PUBLIC setMachineError : booL
VAR_INPUT
END_VAR
END_METHOD

METHOD PUBLIC stateComplete : BOOL //Result = TRUE if state completed (BusyIntern=TRUE)
VAR_INPUT
END_VAR
END_METHOD

{attribute 'monitoring' := 'call'}
PROPERTY public actMode : eMODE
GET
END_GET
END_PROPERTY

{attribute 'monitoring' := 'call'}
//Actual state enum, only read access by default, check options for further options 
PROPERTY public actState : eSTATE
GET
END_GET
SET
END_SET
END_PROPERTY

{attribute 'monitoring' := 'call'}
PROPERTY isBusy : BOOL
GET
END_GET
END_PROPERTY

PROPERTY PUBLIC setStateComplete : BOOL
GET
END_GET
SET
END_SET
END_PROPERTY

END_INTERFACE

// POUs/Statemodel/UnitTemplate/Statemodel_Unit
{attribute 'no_check'}
//Generic Unit 
FUNCTION_BLOCK Statemodel_Unit implements I_Statemodel_Unit
VAR_OUTPUT CONSTANT
END_VAR             										
VAR_INPUT           										
	unit																:	Statemodel;		
END_VAR             										
VAR_OUTPUT          										
END_VAR             	
VAR                 	
(* Local variables ************************************************************)

(* Trigger *****************************************************************)

(* Timer ******************************************************************)

(* Fcuntion blocks ***************************************************************)

(* Dummys **********************************************************)

END_VAR

	(* Generic unit incl. state model										V1.0		*)
	(************************************************************************************)

(* work local sub ****************************************)
	Unit();
	IF Unit.RT_StateChanged THEN stateChanged(unit.Mode, Unit.State); END_IF
	
(* call methods ********************************************)
	CASE Unit.state OF
	eSTATE.STARTUP			:	Startup();
	eSTATE.IDLE				: 	Idle();
	eSTATE.STARTING			:	Starting();		
	eSTATE.STARTED			: 	Started();	
	eSTATE.EXECUTE			:	Executing();
	eSTATE.COMPLETING		:	Completing();
	eSTATE.COMPLETE			: 	Complete();
	eSTATE.ABORTING			:	Aborting();
	eSTATE.ABORTED			:  	Aborted();
	eSTATE.CLEARING			:	Clearing();
	eSTATE.STOPPING			:	Stopping();
	eSTATE.STOPPED			: 	Stopped();
	eSTATE.RESETTING		:	Resetting();
	ELSE
		;
	END_CASE

(*********************************************************)

METHOD PROTECTED aborted : BOOL
VAR_INPUT
END_VAR
Aborted														:= unit.InAborted;
END_METHOD

METHOD PROTECTED aborting : BOOL
VAR_INPUT
END_VAR
Unit.StateComplete();
Aborting													:= Unit.InAborting;
END_METHOD

METHOD PROTECTED clearing : Bool
VAR_INPUT
END_VAR
Unit.StateComplete();
Clearing													:= Unit.InClearing;
END_METHOD

METHOD PROTECTED complete : Bool
VAR_INPUT
END_VAR
Complete														:= unit.InComplete;
END_METHOD

METHOD PROTECTED completing : BOOL
VAR_INPUT
END_VAR
Unit.StateComplete();
Completing													:= Unit.InCompleting;
END_METHOD

METHOD PROTECTED executing : booL
VAR_INPUT
END_VAR
Executing 												:= Unit.InExecute;
END_METHOD

METHOD FB_exit : BOOL
VAR_INPUT
	bInCopyCode : BOOL; // if TRUE, the exit method is called for exiting an instance that is copied afterwards (online change).
END_VAR
FB_EXit															:= TRUE;
END_METHOD

METHOD FB_init : BOOL
VAR_INPUT
	bInitRetains : BOOL; // if TRUE, the retain variables are initialized (warm start / cold start)
	bInCopyCode : BOOL;  // if TRUE, the instance afterwards gets moved into the copy code (online change)
END_VAR
(* Example 
	Unit.pSubRemoteData[1]												:= ADR(Infeed.unit.RemoteData);
	Unit.pSubRemoteData[2]												:= ADR(Support_1.unit.RemoteData);
	Unit.pSubRemoteData[3]												:= ADR(Support_2.RemoteData);	
	Unit.pSubRemoteData[4]												:= ADR(Transport.unit.RemoteData);
	Unit.pSubRemoteData[5]												:= ADR(Outfeed.unit.RemoteData);
*)
FB_init														:= TRUE;
END_METHOD

METHOD FB_reinit : BOOL
VAR_INPUT
END_VAR
FB_reinit											:= TRUE;
END_METHOD

METHOD PROTECTED idle : Bool
VAR_INPUT
END_VAR
Idle														:= unit.InIdle;
END_METHOD

METHOD PROTECTED Resetting : Bool
VAR_INPUT
END_VAR
Unit.StateComplete();
Resetting													:= Unit.InResetting;
END_METHOD

{attribute 'monitoring' := 'call'}
PROPERTY public rUnit : REFERENCE TO Statemodel
GET
rUnit REF= Unit;
END_GET
END_PROPERTY

METHOD PROTECTED started : Bool
VAR_INPUT
END_VAR
Started													:= Unit.InStarted;
END_METHOD

METHOD PROTECTED starting : Bool
VAR_INPUT
END_VAR
Unit.StateComplete();
Starting													:= Unit.InStarting;
END_METHOD

METHOD PROTECTED startup : Bool
VAR_INPUT
END_VAR
Unit.StateComplete();
Startup													:= Unit.InStartup;
END_METHOD

METHOD PROTECTED stateChanged : BOOL 
VAR_INPUT
	mode											:	eMODE;
	state											:	eSTATE;
END_VAR
END_METHOD

METHOD PROTECTED stopped : Bool
VAR_INPUT
END_VAR
Stopped														:= unit.InStopped;
END_METHOD

METHOD PROTECTED stopping : Bool
VAR_INPUT
END_VAR
Unit.StateComplete();
Stopping													:= Unit.InStopping;
END_METHOD

END_FUNCTION_BLOCK

// POUs/Statemodel/UnitTemplate/I_Statemodel_Unit
INTERFACE I_Statemodel_Unit Extends __System.IQueryInterface

{attribute 'monitoring' := 'call'}
PROPERTY public rUnit : REFERENCE TO Statemodel
GET
END_GET
END_PROPERTY

END_INTERFACE

// POUs/Motion/TF50xx-NC/03_Utilities/CoordinateTransformation2D
FUNCTION_BLOCK CoordinateTransformation2D //CoordinateTransformation
// transformation of an X/Y product coordinate to the machine coordinate system
// MCS = machine coordinate system
// PCS = product coordinate system
VAR_INPUT
//Parameter
	x0 														: LREAL;		// origin MCS X coordinate of the product coordinate system
	y0 														: LREAL;		// origin MCS Y coordinate of the product coordinate system
	x1 														: LREAL;		// opposite corner point MCS X coordinate of the product 
	y1 														: LREAL;		// opposite corner point MCS Y coordinate of the product
	a 														: LREAL;		// length of the product (difference x1pcs-x0pcs)
	b 														: LREAL;		// width of the product (difference y1pcs-y0pcs)
END_VAR                                                 	
VAR_OUTPUT                                              	
	Xmcs 													: LREAL;	// X coordinate in machine coordinate system
	Ymcs 													: LREAL;	// Y coordinate in machine coordinate system
															
	Xpcs 													: LREAL;	// X coordinate in Product coordinate system
	Ypcs 													: LREAL;	// Y coordinate in Product coordinate system
                                                        	
	Alfa													: LREAL;	

	Error 													: BOOL;	
//		ErrorID 											: UDINT;
END_VAR
VAR
	c														: LREAL;
	diagonal												: LREAL;

	ratio													: LREAL;
	
	alfa1													: LREAL;
	alfa2													: LREAL;
END_VAR

;

{attribute 'monitoring' := 'call'}
PROPERTY PUBLIC diagonalMSC : LREAL
GET
VAR
	t		:	LREAL;
END_VAR
t 			:=  EXPT(X1-X0,2.0) + EXPT(y1-y0,2.0);
DiagonalMSC := SQRT(t);
END_GET
END_PROPERTY

{attribute 'monitoring' := 'call'}
PROPERTY PUBLIC diagonalPCS : LREAL
GET
DiagonalPCS := SQRT((a*a)+(b*b));
END_GET
END_PROPERTY

{attribute 'monitoring' := 'call'}
PROPERTY PUBLIC isParamValid : BOOL
GET
IsParamValid 													:= not ParamHasError;
END_GET
SET
PUBLIC 
VAR
END_VAR
IF NOT IsParamValid
THEN
	a 														:= 0.0;
	b 														:= 0.0;
	x1 														:= Y1 := 0.0;
	y0 														:= X0 := 0.0;
END_IF
END_SET
END_PROPERTY

METHOD MSCtoPCS : BOOL //Return value = TRUE if execution finished successful / FALSE if finished with error
VAR_INPUT
	Xmcs 													: LREAL;	// X coordinate in machine coordinate system
	Ymcs 													: LREAL;	// Y coordinate in machine coordinate system
END_VAR
IF ParamHasError THEN
	Error 													:= TRUE; 
	MSCtoPCS 												:= FALSE;
ELSE	
	THIS^.Xmcs												:= Xmcs;	
	THIS^.Ymcs												:= Ymcs;	

	c 														:= SQRT(a*a + b*b);
	alfa 													:= ACOS((x1-x0) / c) - ACOS( a / c);
	
	Xpcs 													:= 	 (Xmcs - x0) * COS(alfa) + (Ymcs - y0) * SIN(alfa);
	Ypcs 													:= - (Xmcs - x0) * SIN(alfa) + (Ymcs - y0) * COS(alfa);
	
	Error 													:= FALSE; 
	MSCtoPCS 												:= TRUE;
END_IF
END_METHOD

{attribute 'monitoring' := 'call'}
PROPERTY PRIVATE paramHasError : BOOL
GET
ParamHasError := 	a<=0.0 
			OR 	b<=0.0 
			OR 	x1=x0 
			OR 	y1=y0;
END_GET
END_PROPERTY

METHOD PUBLIC PCStoMSC : booL //Return value = TRUE if execution finished successful / FALSE if finished with error
VAR_INPUT
	Xpcs : LREAL;	// X coordinate in product coordinate system
	Ypcs : LREAL;	// Y coordinate in product coordinate system	
END_VAR
IF ParamHasError 
THEN
	Error 													:= TRUE; 
	PCStoMSC												:= FALSE;
ELSE                										
	THIS^.Xpcs												:= Xpcs;	
	THIS^.Ypcs												:= Ypcs;
	
	c 														:= SQRT(a*a + b*b);
	diagonal												:= SQRT((x1-x0)*(x1-x0)+(y1-y0)*(y1-y0));
	
	ratio													:= diagonal/c;
	
	alfa1 													:= ACOS((x1-x0) / diagonal);
	alfa2													:= ACOS(a/c);
	
	alfa													:= alfa1-alfa2;
	
	Xmcs 													:= x0 + ratio * (Xpcs * COS(alfa) - Ypcs * SIN(alfa));
	Ymcs 													:= y0 + ratio * (Xpcs * SIN(alfa) + Ypcs * COS(alfa));
                    	
	Error 													:= FALSE; 
	PCStoMSC												:= TRUE;
END_IF
END_METHOD

END_FUNCTION_BLOCK

// POUs/Motion/TF50xx-NC/03_Utilities/getOvrVelo
{attribute 'no_check'}
//Overwrite function - Returns velocity setpoint based on max velo and requested overwrite 
FUNCTION getOvrVelo : LREAL
VAR_INPUT
	SetVelo													:	LREAL;
	MaxVelo													:	LREAL;
END_VAR
VAR
END_VAR

IF 	MaxVelo = 0.0 OR SetVelo = 0.0
THEN
	GetOvrVelo 												:= 0.0;
ELSE                										
	GetOvrVelo 												:= 100.0 / MaxVelo * SetVelo;
END_IF

END_FUNCTION

// POUs/Motion/TF50xx-NC/AxNcBase
FUNCTION_BLOCK AxNcBase EXTENDS AXIS_REF IMPLEMENTS I_AxNcBase(* See Tc2_MC2 *)
VAR_OUTPUT CONSTANT
	OPTION_EN_CMD_ABORTED_ERROR								: 	BYTE := 2#1000_0000; //Default: .7 = xxx.CmdAborted is treaded as error
END_VAR
VAR_INPUT
{attribute 'displaymode':='binary'}
	Options													: 	BYTE  := OPTION_EN_CMD_ABORTED_ERROR; //See output constant for Options mask
	
(* Axis *)
	Admin													: 	AxAdmin;
	para													: 	AxPara;

	Home													:	AxHoming;
	event													:	AxEventHandling;                                                   
END_VAR                                             	
VAR_OUTPUT                                          	
	ErrHdl													:	ERROR_HDL;
END_VAR
VAR
END_VAR

	(* Axis 																*)
	(************************************************************************)

	
(********************************************************************************)
(* Error NC																		*)
(********************************************************************************)
	Event(
		Enable		:= Admin.EnableOK OR Event.NoOfActiveEvents > 0,
		ConfirmTrig	:= Admin.ResetTrig,
		Name		:= para.Name,
		SourceId	:= (* Default *) ,
		rAxis		:= THIS^,
		ErrorId		:= TO_UDINT(ErrHdl.Id),
		Status		=> );
		
	(* Init ErrHdl *)
	ErrHdl.Reset();

(********************************************************************************)
(* work Admin ctrl 																*)
(********************************************************************************)
	Admin(rAxis		:= THIS^);
	IF Admin.Error
	THEN
		ErrHdl.id 											:= UDINT_TO_DINT(Admin.ErrorId);
		ErrHdl.fnc											:= 'Admin';
		ErrHdl.text											:= Admin.ErrorText;
		ErrHdl.flag											:= TRUE;
	END_IF
	
(********************************************************************************)
(* Parameter																	*)
(********************************************************************************)
	para(Axisid := NcToPlc.AxisId);
		
(********************************************************************************)
(* work homing ctrl 															*)
(********************************************************************************)
	Home(rAxis := THIS^ );
	errorCheck(AxBase := Home);
	

(********************************************************************************)

METHOD PROTECTED errorCheck : BOOL
VAR_IN_OUT
	AxBase									:	AxFbBase;
END_VAR
IF AxBase.Error
THEN
	ErrHdl.flag									:= TRUE;
	ErrHdl.fnc									:= 'AxNcPtP';
	ErrHdl.id									:= TO_DINT(AxBase.ErrorID);
	ErrHdl.text									:= AxBase.ErrorText;
	errorCheck									:= TRUE;
ELSIF AxBase.CmdAborted AND Options.7
THEN
	ErrHdl.id 									:= 19200;
	ErrHdl.fnc									:= 'AxNcPtP';
	ErrHdl.text									:= 'command aborted';
	ErrHdl.flag									:= TRUE;		
ELSE
	errorCheck									:= FALSE;
END_IF
END_METHOD

METHOD PUBLIC noAction : BOOL //Return value = TRUE if busy of home and motion 
VAR_INPUT
END_VAR
home.Execute	:= FALSE;


NoAction 		:= 	NOT home.Busy ;
END_METHOD

PROPERTY PUBLIC optEnableCmdAbortedAsError : BOOL
GET
optEnableCmdAbortedAsError := Options.7;
END_GET
SET
Options.7 := optEnableCmdAbortedAsError;
END_SET
END_PROPERTY

{attribute 'monitoring' := 'call'}
PROPERTY rAdmin : REFERENCE to AxAdmin
GET
rAdmin REF= Admin;
END_GET
END_PROPERTY

{attribute 'monitoring' := 'call'}
PROPERTY rAxisRef : REFERENCE TO AXIS_REF
GET
rAxisRef REF= THIS^;
END_GET
END_PROPERTY

{attribute 'monitoring' := 'call'}
PROPERTY PUBLIC rErrHdl : REFERENCE to ERROR_HDL
GET
rErrHdl REF= ErrHdl;
END_GET
SET
ErrHdl := rErrHdl;
END_SET
END_PROPERTY

METHOD reset : Bool
VAR_INPUT
END_VAR
NoAction();
reset 			:= ErrHdl.flag OR Admin.reset(FALSE);
Event.confirm();
END_METHOD

{attribute 'monitoring' := 'call'}
PROPERTY rHome : REFERENCE To AxHoming
GET
rHome REF= Home;
END_GET
END_PROPERTY

{attribute 'monitoring' := 'call'}
PROPERTY rPara : REFERENCE TO AxPara
GET
rPara REF= Para;
END_GET
END_PROPERTY

END_FUNCTION_BLOCK

// POUs/Motion/TF50xx-NC/AxNcPTP
FUNCTION_BLOCK AxNcPTP EXTENDS AxNcBase implements I_AxNcPTP (* See Tc2_MC2 *)
VAR_OUTPUT CONSTANT
END_VAR
VAR_INPUT
	Motion													:	AxMotion;                                        
END_VAR                           
VAR_OUTPUT                  	
END_VAR
VAR

END_VAR

	(* Axis 																*)
	(************************************************************************)

	
(********************************************************************************)
(* Call AxNcBase																*)
(********************************************************************************)
	Super^();
		
(********************************************************************************)
(* work moving ctrl 															*)
(********************************************************************************)
	Motion(rAxis := THIS^);
	errorCheck(AxBase := Motion);
	
(********************************************************************************)

METHOD PUBLIC noAction : BOOL //Return value = TRUE if busy of home and motion 
VAR_INPUT
END_VAR

Motion.Execute	:= FALSE;
Motion.JogBwd	:= FALSE;
Motion.JogFwd	:= FALSE;

NoAction 		:= 	Super^.noAction() and NOT Motion.Busy;
END_METHOD

{attribute 'monitoring' := 'call'}
PROPERTY rMotion : REFERENCE TO AxMotion
GET
rMotion REF= Motion;
END_GET
END_PROPERTY

END_FUNCTION_BLOCK

// POUs/Motion/TF50xx-NC/AxNcBaseExt
FUNCTION_BLOCK AxNcBaseExt EXTENDS AxNcBase 
VAR_OUTPUT CONSTANT
END_VAR
VAR_INPUT
	State													:	AxStatemodel;                                               
END_VAR                                             	
VAR_OUTPUT                                          	
END_VAR
VAR
END_VAR

	(* Axis 																*)
	(************************************************************************)

	
(********************************************************************************)
(* Call super 																	*)
(********************************************************************************)
	SUPER^();

(********************************************************************************)
(* Execute unit state model														*)
(********************************************************************************)
	State(
		Unit						:=  ,
		rAxis						:= THIS^,
		ENDisableInAborting			:= ,
		SafetyOK					:= ,//NOT Drive.SafetyError,
		ErrorActive					:= Event.ErrorId <> 0);

	//Execute aller Bausteine zuruecknehmen
	IF state.unit.InResetting 
		AND State.unit.RT_StateChanged
	THEN
		NoAction();
	END_IF

(********************************************************************************)

END_FUNCTION_BLOCK

// POUs/Motion/TF50xx-NC/AxNcPtpGear
FUNCTION_BLOCK AxNcPtpGear EXTENDS AxNcPTP
VAR_OUTPUT CONSTANT
END_VAR
VAR_INPUT
(* Axis *)
	Gear													:	AxGear;                                                
END_VAR                                             	
VAR_OUTPUT                                          	
END_VAR
VAR
END_VAR

	(* Axis extended (Incl. Gearing)										*)
	(************************************************************************)
	
(********************************************************************************)
(* work basic	 																*)
(********************************************************************************)
	SUPER^();

(********************************************************************************)
(* work gear ctrl 																*)
(********************************************************************************)
	gear(rAxis := THIS^);
	errorCheck(AxBase := Gear);
	
(********************************************************************************)

METHOD PUBLIC noAction : BOOL //Return value = TRUE if busy of home and motion 
VAR_INPUT
END_VAR
Gear.Execute	:= FALSE;

NoAction 		:= 	SUPER^.NoAction() AND NOT Gear.Busy ;
END_METHOD

METHOD reset : Bool
VAR_INPUT
END_VAR
Gear.Execute		:= FALSE;
reset 				:= SUPER^.reset();
END_METHOD

END_FUNCTION_BLOCK

// POUs/Motion/TF50xx-NC/AxNcPTPwJobs
FUNCTION_BLOCK AxNcPTPwJobs EXTENDS AxNcPTP (* See Tc2_MC2 *)
VAR_OUTPUT CONSTANT
	MIN_JOB													:	INT := 0;
	MAX_JOB													:	INT := 5;
	
{attribute 'displaymode':='binary'}
	OPTION_EN_CYCLIC_TARGET_CHECK							: 	BYTE := 2#0000_0001; //.0 = Cyclic target check	
END_VAR
VAR_INPUT
	Job														:	ARRAY[MIN_JOB..MAX_JOB] OF AX_JOB;	                              
END_VAR                           
var_output                  	
	JobId													:	INT := MIN_JOB;
END_VAR
VAR
	i 														: 	INT;
END_VAR

	(* Axis 																*)
	(************************************************************************)

	
(********************************************************************************)
(* Call AxNcBase																*)
(********************************************************************************)
	Super^();
			
(* Check start arr pos **********************************************************)
	IF Options.0 AND Para.InitDone THEN	CheckTargetPos(); END_IF
	
(********************************************************************************)

METHOD PUBLIC checkTargetPos : INT //ID of last job which is in target / 0 if no job is in target
VAR_INPUT
END_VAR
CheckTargetPos				:= 0;
FOR i := MIN_JOB TO MAX_JOB DO
	IF Job[i].Fnc = 6 THEN
		Job[i].InTarget := Status.NotMoving
									AND(
									NcToPlc.ModuloActPos >= Job[i].Target - para.TargetPosWindow
									AND NcToPlc.ModuloActPos <= Job[i].Target + para.TargetPosWindow
									OR
									(MODABS(Job[i].Target,para.ModuloFactor) <= 0 + para.TargetPosWindow
									OR MODABS(Job[i].Target,para.ModuloFactor) >= para.ModuloFactor - para.TargetPosWindow)
									AND(
									NcToPlc.ModuloActPos >= para.ModuloFactor - para.TargetPosWindow
									OR NcToPlc.ModuloActPos <= 0 + para.TargetPosWindow));

		Job[i].InPosWindow	:= NcToPlc.ModuloActPos >= Job[i].Target - para.PosRangeWindow
									AND NcToPlc.ModuloActPos <= Job[i].Target + para.PosRangeWindow
									OR
									(MODABS(Job[i].Target,para.ModuloFactor) <= 0 + para.PosRangeWindow
									OR MODABS(Job[i].Target,para.ModuloFactor) >= para.ModuloFactor - para.PosRangeWindow)
									AND(
									NcToPlc.ModuloActPos >= para.ModuloFactor - para.PosRangeWindow
									OR NcToPlc.ModuloActPos <= 0 + para.PosRangeWindow);
	ELSE
		Job[i].InTarget := Status.NotMoving
									AND NcToPlc.ActPos >= Job[i].Target - para.TargetPosWindow
									AND NcToPlc.ActPos <= Job[i].Target + para.TargetPosWindow ;

		Job[i].InPosWindow	:= NcToPlc.ActPos >= Job[i].Target - para.PosRangeWindow
									AND NcToPlc.ActPos <= Job[i].Target + para.PosRangeWindow;
	END_IF
	
	IF Job[i].InTarget 
	THEN
		CheckTargetPos		:= i;
	END_IF
END_FOR
END_METHOD

PROPERTY PUBLIC optEnableCyclicCheckTargetPos : BOOL
GET
optEnableCyclicCheckTargetPos := Options.0;
END_GET
SET
Options.0 := optEnableCyclicCheckTargetPos;
END_SET
END_PROPERTY

METHOD PUBLIC startMotion : BOOL
VAR_INPUT
	Execute			:	BOOL;
	JobID			:	int ;
END_VAR
THIS^.JobID		:= Jobid;

IF JobID >= MIN_JOB AND JobId <= MAX_JOB
THEN
	CheckTargetPos();
//	startName				:= Job[Jobid].name;
	Motion.Fnc 				:= Job[Jobid].Fnc;
	Motion.BufferMode 		:= Job[Jobid].BufferMode;
	Motion.Direction 		:= Job[Jobid].Direction;
	Motion.Target 			:= Job[Jobid].Target;
	Motion.Velo 			:= Job[Jobid].Velo;
	Admin.Override 			:= Job[Jobid].Override;
	Motion.Acc		 		:= Job[Jobid].Acc;
	Motion.Dec				:= Job[Jobid].Dec;
	Motion.Jerk	 			:= Job[Jobid].Jerk;
	MOtion.Execute			:= Execute;
	StartMotion				:= TRUE;
ELSE
	StartMotion				:= FALSE;
END_IF
END_METHOD

END_FUNCTION_BLOCK

// POUs/Motion/TF5100-NCI/01_Main/NCI_REF
{attribute 'no_check'}
FUNCTION_BLOCK NCI_REF
VAR_INPUT
	PlcToNci										AT %Q*	: PLCTONC_NCICHANNEL_REF;	//link PLC to NC
END_VAR                             				
VAR_OUTPUT                          	
	NciToPlc										AT %I*	: NCTOPLC_NCICHANNEL_REF;	//link NC to PLC

(* Extrabits out of the struct *)
	ItpRunning												:	BOOL := FALSE;	//Interpreter is running
	ItpGroupActive											:	BOOL;			//Interpreter group is active -> Axes group build 			
	GrpCnfg													:	NCI_EXT3DGROUP;	//Group configuration
	                                    					
(* ChnState *******************)        					
	IsItpChn												:	BOOL := FALSE;	//TRUE when it is interpreter channel
	IsEStopRequested										:	BOOL := FALSE;	//TRUE when EStop is requested
	IsFeedFromBackupList									:	BOOL := FALSE;	//TRUE when parameter feed comes from backup list 
	IsMovingBackward										:	BOOL := FALSE;	//TRUE when moving forward
	
(* configurated parameters of the cyclic channel *)
	PathRestWay												:	LREAL;	//remaining arc length on the current path segment
	CurrentPathSetVelo										:	LREAL;	//current path set velocity
                                        					
	SAFStatus												:	UDINT;	//SAF state
	SAFEintraege											:	UDINT;	//current number of SAF entries/tasks
	SVBStatus												:	UDINT;	//SVB state
	SVBEintraege											:	UDINT;	//current number of SVB entries/tasks
	MemLastBlockNo											:	UDINT;	//contains last block number
END_VAR
VAR
	(* NciToPlc channel extend *)
	SetCyclicLrealOffsets									:	ItpSetCyclicLRealOffsets;
	SetCyclicLrealOffsetsDone								:	BOOL;
	SetCyclicUdintOffsets									:	ItpSetCyclicUdintOffsets;
	SetCyclicUdintOffsetsDone								:	BOOL;
	
END_VAR

;

METHOD readStatus : BOOL 
VAR_INPUT
END_VAR
(* NCI Status lesen															*)
(****************************************************************************)

(****************************************************************************)
(* 4 LReal variables to configurate the interface cyclely					*)
(****************************************************************************)
	IF SetCyclicLRealOffsets.bExecute AND NOT SetCyclicLRealOffsets.bBusy
	THEN
		SetCyclicLRealOffsetsDone := NOT SetCyclicLRealOffsets.bErr;
	END_IF

	IF NOT SetCyclicLRealOffsetsDone
	THEN
		SetCyclicLRealOffsets(
			bExecute			:= NciToPlc.ChnId <> 0 AND NOT SetCyclicLRealOffsetsDone AND NOT SetCyclicLRealOffsets.bErr,
			tTimeOut			:= DEFAULT_ADS_TIMEOUT,
			nIndexOffsetParam1	:= 16#500, (* Bahnrestweg (verbleibende Bogenlaenge) auf dem aktuellen Bahnsegment *)
			nIndexOffsetParam2	:= 16#502 , (* aktuelle Bahnsollgeschwindigkeit *)
			nIndexOffsetParam3	:= ,
			nIndexOffsetParam4	:= ,
			sNciToPlc			:= NciToPlc,
			bBusy				=> ,
			bErr				=> ,
			nErrId				=> );
	END_IF

	(* reading date *)
	PathRestWay												:= NciToPlc.DoubleParams[0];	
	CurrentPathSetVelo										:= NciToPlc.DoubleParams[1];	
	//														:= NciToPlc.DoubleParams[2];	
	//														:= NciToPlc.DoubleParams[0];	

(******************************************************************************)
(* 4 DINT variables cycliaclly das Zyklsiche Interface konfigurieren						*)
(******************************************************************************)
	IF SetCyclicUdintOffsets.bExecute 
	AND NOT SetCyclicUdintOffsets.bBusy
	THEN
		SetCyclicUdintOffsetsDone 							:= NOT SetCyclicUdintOffsets.bErr;
	END_IF

	IF NOT SetCyclicUdintOffsetsDone
	THEN
		SetCyclicUdintOffsets(
			bExecute			:= NciToPlc.ChnId <> 0 AND NOT SetCyclicUdintOffsetsDone AND NOT SetCyclicUdintOffsets.bErr,
			tTimeOut			:= DEFAULT_ADS_TIMEOUT,
			nIndexOffsetParam1	:= 16#4, (* Akt SVB Status 4  *)
			nIndexOffsetParam2	:= 16#5, (* Akt SAF Status -> Running 5 *)
			nIndexOffsetParam3	:= 16#B, (* Akt Anzahl SVB Eintraege B *)
			nIndexOffsetParam4	:= 16#C, (* Akt Anzahl SAF Eintraege C *)
			sNciToPlc			:= NciToPlc,
			bBusy				=> ,
			bErr				=> ,
			nErrId				=> );
	END_IF	

	(* Daten lesen *)
	SVBStatus												:= NciToPlc.IntParams[0];	
	SAFStatus												:= NciToPlc.IntParams[1];	
	SVBEintraege											:= NciToPlc.IntParams[2];	
	SAFEintraege											:= NciToPlc.IntParams[3];	
	
(******************************************************************************)
(* Interpreterstatus lesen																		*)
(******************************************************************************)
	ItpRunning 												:= NciToPlc.ItpState > NCI_INTERPRETER_READY
																	AND NciToPlc.ItpState <> NCI_INTERPRETER_ABORTED
																	OR SAFStatus > 2
																	OR SVBStatus > 2
																	OR SAFEintraege > 0
																	OR SVBEintraege > 0;
                                							
	IF NciToPlc.BlockNo > 0 
	AND MemLastBlockNo <> NciToPlc.BlockNo
	THEN
		MemLastBlockNo 	 									:= NciToPlc.BlockNo;
	END_IF                      							
	                            							
	GrpCnfg.nXAxisId										:= NciToPlc.AcsAxisIDs[0];
	GrpCnfg.nYAxisId										:= NciToPlc.AcsAxisIDs[1];
	GrpCnfg.nZAxisId										:= NciToPlc.AcsAxisIDs[2];
	GrpCnfg.nQ1AxisId										:= NciToPlc.AcsAxisIDs[3];
	GrpCnfg.nQ2AxisId										:= NciToPlc.AcsAxisIDs[4];
	GrpCnfg.nQ3AxisId										:=	NciToPlc.AcsAxisIDs[5];
	GrpCnfg.nQ4AxisId										:= NciToPlc.AcsAxisIDs[6];
	GrpCnfg.nQ5AxisId										:= NciToPlc.AcsAxisIDs[7];
                                							
	ItpGroupActive											:= GrpCnfg.nXAxisId <> 0
																	OR GrpCnfg.nYAxisId <> 0
																	OR GrpCnfg.nZAxisId <> 0
																	OR GrpCnfg.nQ1AxisId <> 0
																	OR GrpCnfg.nQ2AxisId <> 0
																	OR GrpCnfg.nQ3AxisId <> 0
																	OR GrpCnfg.nQ4AxisId <> 0
																	OR GrpCnfg.nQ5AxisId <> 0;
                                	
(******************************************************************************)
(* Channelstatus lesen																			*)
(******************************************************************************)
	IsItpChn												:= NciToPlc.ChnState.0;
	IsEStopRequested										:= NciToPlc.ChnState.8;
	IsFeedFromBackupList									:= NciToPlc.ChnState.10;
	IsMovingBackward										:= NciToPlc.ChnState.11;

	
(* ENUM ItpMode
	0x0	Defaultbelegung (Abwahl der übrigen Betriebsarten)
	0x1	Einzelsatzbetrieb im NC-Kern (Satzausführungstask/SAF)
	0x1000	reserviert
	0x2000	reserviert
	0x4000	Einzelsatzbetrieb im Interpreter
*)

(* ItpStatus
ITP_STATE_IDLE  The interpreter is in idle state when there is no NC program loaded as yet or when a group reset is being executed.
The interpreter also goes into idle state when a current program is stopped. In the case a group reset must be executed in order to prevent error 0x42C5. 
It is therefore recommended to execute a group reset after stopping via the PLC.
 
ITP_STATE_READY  After successful loading of an NC program, the interpreter is in ready state.
After a program has been successfully processed and exited, the interpreter goes into ready state. 
In the meantime, however, other states are accepted.  
 
ITP_STATE_ABORTED  Tritt während der Abarbeitung des NC Programms ein Laufzeitfehler auf, 
so geht der Interpreter in den Aborted eSTATE. Der eigentliche Fehlercode ist dem Kanal Status zu entnehmen.  

ITP_STATE_SINGLESTOP  If a run time error occurs during the processing of an NC program, the interpreter goes into aborted state. The actual error code is given in Channel Status.
 
NCI_INTERPRETER_INITFAILED:	UDINT	:=	0;
NCI_INTERPRETER_IDLE:			UDINT	:=	1;
NCI_INTERPRETER_READY:			UDINT	:=	2;
NCI_INTERPRETER_STARTED:		UDINT	:=	3;
NCI_INTERPRETER_SCANNING:		UDINT	:=	4;
NCI_INTERPRETER_RUNNING:		UDINT	:=	5;
NCI_INTERPRETER_STAY_RUNNING:	UDINT	:=	6;
NCI_INTERPRETER_WRITETABLE:		UDINT	:=	7;
NCI_INTERPRETER_SEARCHLINE:		UDINT	:=	8;
NCI_INTERPRETER_END:			UDINT	:=	9;
NCI_INTERPRETER_SINGLESTOP:		UDINT	:=	10;
NCI_INTERPRETER_ABORTING:		UDINT	:=	11;
NCI_INTERPRETER_ABORTED:		UDINT	:=	12;
NCI_INTERPRETER_FAULT:			UDINT	:=	13;
NCI_INTERPRETER_RESET:			UDINT	:=	14;
NCI_INTERPRETER_STOP:			UDINT := 15;
NCI_INTERPRETER_WAITFUNC:		UDINT	:=	16;
NCI_INTERPRETER_FLUSHBUFFERS:	UDINT	:=	17;

*)

	readStatus											:= TRUE;
(******************************************************************)
END_METHOD

END_FUNCTION_BLOCK

// POUs/Motion/TF5100-NCI/01_Main/NciAdmin
{attribute 'no_check'}
//NCI group administration - Build/Reconfig group via Enable input, activate EStop and StepOn after releasing EStop input
//based on Tc2_NCI library
FUNCTION_BLOCK NciAdmin
VAR_INPUT
	ResetAdmin												:	BOOL := FALSE; (* Reset Nci group *)
	Enable													:	BOOL := FALSE; (* TRUE = Build Group / FALSE = Reconfig Group *)
	EStop													:	BOOL := FALSE; (* TRUE = EStop / FALSE = StepOn *)
	SingleBlockMode											:	E_ItpSingleBlockMode := ItpSingleBlockOff; (* Operation mode for single set:
																											 	ItpSingleBlockOff: single set off
																											 	ItpSingleBlockNck: single set in the NC kernel 
																												ItpSingleBlockIntp: single set in the interpreter *)
	InSingleBlockTrigNext									:	BOOL	:= FALSE;
	GrpCnfg													:	NCI_EXT3DGROUP;
	Override												:	LREAL := 0.0; //0.0-100.0%
	SpindleOvr												:	LREAL := 0.0; //0.0-100.0%
	rNCIRef													:	REFERENCE TO NCI_REF := 0;
END_VAR
VAR_IN_OUT
END_VAR
VAR_OUTPUT
	InGroup													:	BOOL; 
	Busy													:	BOOL;
	Done													:	BOOL;
	Error													:	BOOL;
{attribute 'displaymode':='hex'}
	ErrorID													:	UDINT;
	ErrorText												:	STRING(40);
END_VAR
VAR
(* Zwischenspeicher **************************************************************************)
	MemDone													:	BOOL;
	MemFnc													:	INT := 0;

(* Instanzierung der MC Bausteine *******************************************************)
	ItpSingleBlock											:	ItpSingleBlock := (tTimeOut	:= DEFAULT_ADS_TIMEOUT);
	CfgBuildExt3DGroup										:	CfgBuildExt3DGroup := (tTimeOut	:= DEFAULT_ADS_TIMEOUT);
	CfgReconfigGroup										:	CfgReconfigGroup := (tTimeOut	:= DEFAULT_ADS_TIMEOUT);
	ItpResetEx2												:	ItpResetEx2 := (tTimeOut	:= DEFAULT_ADS_TIMEOUT);
	ItpEStopEx												:	ItpEStopEx := (tTimeOut	:= DEFAULT_ADS_TIMEOUT);
	ItpStepOnAfterEStopEx									:	ItpStepOnAfterEStopEx := (tTimeOut	:= DEFAULT_ADS_TIMEOUT);

(* Dummy  **********************************************************)
	Dummy 	: BOOL;
END_VAR

	(* NCI group administration															*)
	(************************************************************************************)

(* verify reference ***********************************************************************)
IF NOT __ISVALIDREF(rNCIRef) 
THEN
	Busy													:= NOT Error;
	ErrorId													:= E_AdsErr.DEVICE_INVALIDPARM;
	Error													:= TRUE;
	Done													:= FALSE;
	InGroup													:= FALSE;
	ErrorText												:= 'Reference to rNCIRef invalid (0)';
	RETURN;
END_IF

(* reading axis-status from NCtoPLC-channel *************************************************)
	rNCIRef.ReadStatus();

(* writing override into the NC-interface ***************************************************)
	rNCIRef.PlcToNci.ChnAxesOvr 							:= LREAL_TO_DWORD(LIMIT(0.0,Override,100.0) * 10000.0 );
	rNCIRef.PlcToNci.ChnSpindleOvr							:= LREAL_TO_DWORD(LIMIT(0.0,SpindleOvr,100.0) * 10000.0 );

(* Build Grp / rebuild grp ******************************************************************)
	InGroup													:=  NOT CfgBuildExt3DGroup.bBusy AND NOT CfgReconfigGroup.bBusy
																AND(rNCIRef.NciToPlc.AcsAxisIDs[0] = GrpCnfg.nXAxisId 		
																AND rNCIRef.NciToPlc.AcsAxisIDs[1] = GrpCnfg.nYAxisId 
																and rNCIRef.NciToPlc.AcsAxisIDs[2] = GrpCnfg.nZAxisId 
																and rNCIRef.NciToPlc.AcsAxisIDs[3] = GrpCnfg.nQ1AxisId
																and rNCIRef.NciToPlc.AcsAxisIDs[4] = GrpCnfg.nQ2AxisId
																and rNCIRef.NciToPlc.AcsAxisIDs[5] = GrpCnfg.nQ3AxisId
																and rNCIRef.NciToPlc.AcsAxisIDs[6] = GrpCnfg.nQ4AxisId
																AND rNCIRef.NciToPlc.AcsAxisIDs[7] = GrpCnfg.nQ5AxisId																
																OR  
																rNCIRef.NciToPlc.McsAxisIDs[0] = GrpCnfg.nXAxisId 
																AND rNCIRef.NciToPlc.McsAxisIDs[1] = GrpCnfg.nYAxisId 
																and rNCIRef.NciToPlc.McsAxisIDs[2] = GrpCnfg.nZAxisId 
																and rNCIRef.NciToPlc.McsAxisIDs[3] = GrpCnfg.nQ1AxisId
																and rNCIRef.NciToPlc.McsAxisIDs[4] = GrpCnfg.nQ2AxisId
																and rNCIRef.NciToPlc.McsAxisIDs[5] = GrpCnfg.nQ3AxisId
																and rNCIRef.NciToPlc.McsAxisIDs[6] = GrpCnfg.nQ4AxisId
																AND rNCIRef.NciToPlc.McsAxisIDs[7] = GrpCnfg.nQ5AxisId);
							
	Dummy													:= CfgBuildExt3DGroup.bBusy; //Catch busy status before next call of FB
									
	CfgBuildExt3DGroup(
		bExecute	:= Enable AND NOT CfgReconfigGroup.bBusy,
		nGroupId	:= rNCIRef.NciToPlc.GrpId,
		nXAxisId	:= GrpCnfg.nXAxisId,
		nYAxisId	:= GrpCnfg.nYAxisId,
		nZAxisId	:= GrpCnfg.nZAxisId,
		nQ1AxisId	:= GrpCnfg.nQ1AxisId,
		nQ2AxisId	:= GrpCnfg.nQ2AxisId,
		nQ3AxisId	:= GrpCnfg.nQ3AxisId,
		nQ4AxisId	:= GrpCnfg.nQ4AxisId,
		nQ5AxisId	:= GrpCnfg.nQ5AxisId,
		tTimeOut	:= ,
		bBusy		=> ,
		bErr		=> ,
		nErrId		=> );

	IF 	Dummy 
		AND NOT CfgBuildExt3DGroup.bBusy 
		AND NOT CfgBuildExt3DGroup.bErr
	THEN
	//	InGroup												:= TRUE;
		MemDone												:= TRUE;
	END_IF


	(* Reconfig Grp *)
	Dummy													:= CfgReconfigGroup.bBusy;

	CfgReconfigGroup(
		bExecute	:= NOT CfgBuildExt3DGroup.bExecute AND NOT CfgBuildExt3DGroup.bBusy AND InGroup,
		nGroupId	:= rNCIRef.NciToPlc.GrpId,
		tTimeOut	:= ,
		bBusy		=> ,
		bErr		=> ,
		nErrId		=> );

	IF 	Dummy 
		AND NOT CfgReconfigGroup.bBusy 
		AND NOT CfgReconfigGroup.bErr
	THEN
	//	InGroup												:= FALSE;
		MemDone												:= TRUE;
	END_IF


(* Estop ****************************************************************************************)
	Dummy													:= ItpEStopEx.bBusy;

	ItpEStopEx(
		bExecute	:= EStop AND NOT ItpStepOnAfterEStopEx.bBusy,
		fDec		:= (* Dec *),
		fJerk		:= (* Jerk *),
		tTimeOut	:= ,
		sNciToPlc	:= rNCIRef.NciToPlc,
		bBusy		=> ,
		bErr		=> ,
		nErrId		=> );
		
	IF ItpEStopEx.bExecute
	THEN //Triggerd by input
		MemFnc.0											:= TRUE;
	END_IF

	IF 	Dummy 
		AND NOT ItpEStopEx.bBusy 
	THEN
		MemDone												:= NOT ItpEStopEx.bErr;
	END_IF

	(* Step on after estop *)
	Dummy													:= ItpStepOnAfterEStopEx.bBusy;
	
	ItpStepOnAfterEStopEx(
		bExecute	:= NOT ItpEStopEx.bExecute AND NOT ItpEStopEx.bBusy AND rNCIRef.NciToPlc.ChnState.8 AND memFnc.0, //EStopReq ,
		tTimeOut	:= ,
		sNciToPlc	:= rNCIRef.NciToPlc,
		bBusy		=> ,
		bErr		=> ,
		nErrId		=> );

	IF 	Dummy 
		AND NOT ItpStepOnAfterEStopEx.bBusy 
	THEN
		MemDone												:= NOT ItpStepOnAfterEStopEx.bErr;
		MemFnc.0											:= FALSE;
	END_IF
	
(* Method fnc ****************************************************************)
	IF NOT Memfnc.4 
	THEN
		IF ResetAdmin
		THEN			
			MemFnc.4										:= reset(Execute:= TRUE);
		END_IF
	ELSIF NOT reset(Execute:= ResetAdmin)
	THEN
		MemDone												:= TRUE;
		MemFnc.4											:= FALSE;
	END_IF
	
	IF NOT Memfnc.5
	THEN
		IF SingleBlockMode <> ItpSingleBlock.nMode 
		THEN
			MemFnc.5										:= SingleBlockModeChange(Execute:= TRUE,SingleBlockMode := SingleBlockMode);
		END_IF
	ELSIF NOT SingleBlockModeChange(Execute:= FALSE, SingleBlockMode := SingleBlockMode)
	THEN
		MemDone												:= TRUE;
		MemFnc.5											:= FALSE;
	END_IF

	IF NOT Memfnc.6
	THEN
		IF InSingleBlockTrigNext
		THEN
			MemFnc.6										:= SingleBlockTrigNext(Execute:= InSingleBlockTrigNext);
		END_IF
	ELSIF NOT SingleBlockTrigNext(Execute:= InSingleBlockTrigNext)
	THEN
		MemDone												:= TRUE;
		MemFnc.6											:= FALSE;
	END_IF
	
(******************************************************************************)
(* Ctrl Status 																					*)
(******************************************************************************)
	Busy													:= CfgBuildExt3DGroup.bBusy
																OR CfgReconfigGroup.bBusy
																OR ItpResetEx2.bBusy
																OR ItpSingleBlock.bBusy
																OR ItpEStopEx.bBusy
																OR ItpStepOnAfterEStopEx.bBusy;
                            						    	
	Done													:= NOT Busy AND MemDone;
                            						    	
	IF done                 	                        	
	THEN                    	                        	
		MemDone												:= FALSE;
	END_IF                  	                        	
                                                        	
	(* Error Output *)                                  	
	IF Busy                                             	
	THEN                                                	
		Error												:= FALSE;
		ErrorId												:= 0;
		ErrorText											:= '';
	ELSIF CfgBuildExt3DGroup.bErr                       	
		AND CfgBuildExt3DGroup.bExecute                 	
	THEN                                                	
		Error												:= TRUE;
		ErrorId												:= CfgBuildExt3DGroup.nErrID;
		ErrorText											:= CONCAT('CfgBuildExt3DGroup ErrorId: ', UDINT_TO_STRING(Errorid));
                                                        	
	ELSIF CfgReconfigGroup.bErr                         	
		AND CfgReconfigGroup.bExecute                   	
	THEN                                                	
		Error												:= TRUE;
		ErrorId												:= CfgReconfigGroup.nErrID;
		ErrorText											:= CONCAT('CfgReconfigGroup ErrorId: ', UDINT_TO_STRING(Errorid));
                                                        	
	ELSIF ItpEStopEx.bErr                               	
		AND ItpEStopEx.bExecute                         	
	THEN                                                	
		Error												:= TRUE;
		ErrorId												:= ItpEStopEx.nErrID;
		ErrorText											:= CONCAT('ItpEStopEx ErrorId: ', UDINT_TO_STRING(Errorid));
                                                        	
	ELSIF ItpStepOnAfterEStopEx.bErr                    	
		AND ItpStepOnAfterEStopEx.bExecute              	
	THEN                                                	
		Error												:= TRUE;
		ErrorId												:= ItpStepOnAfterEStopEx.nErrID;
		ErrorText											:= CONCAT('ItpStepOnAfterEStopEx ErrorId: ', UDINT_TO_STRING(Errorid));
                                                        	
	ELSIF ItpResetEx2.bErr                              	
		AND ItpResetEx2.bExecute                        	
	THEN                                                	
		Error												:= TRUE;
		ErrorId												:= ItpResetEx2.nErrID;
		ErrorText											:= CONCAT('ItpResetEx2 ErrorId: ', UDINT_TO_STRING(Errorid));
                                    	
	ELSIF ItpSingleBlock.bErr                           	
		AND(ItpSingleBlock.bExecuteModeChange OR ItpSingleBlock.bTriggerNext)            	
	THEN                                                	
		Error												:= TRUE;
		ErrorId												:= ItpSingleBlock.nErrID;
		ErrorText											:= CONCAT('ItpSingleBlock ErrorId: ', UDINT_TO_STRING(Errorid));
                                                        	
	ELSIF rNCIRef.NciToPlc.ErrorCode <> 0               	
	THEN                                                	
		Error												:= TRUE;
		ErrorId												:= rNCIRef.NciToPlc.ErrorCode;
		ErrorText											:= CONCAT('NCI Grp ErrorId: ', UDINT_TO_STRING(Errorid));
	ELSE                    						    	
		Error												:= FALSE;
		ErrorId												:= 0;
		ErrorText											:= '';
	END_IF                  	

(********************************************************************************************************)

METHOD PUBLIC reset : BOOL //Return value = TRUE if busy
//required parameter
//rNCIRef
VAR_INPUT
	Execute													:	BOOL;
END_VAR
IF NOT __ISVALIDREF(rNCIRef) 
THEN
	Busy													:= NOT Error;
	ErrorId													:= E_AdsErr.DEVICE_INVALIDPARM;
	Error													:= TRUE;
	Done													:= FALSE;
	ErrorText												:= 'Reference to rNCIRef invalid (0)';
	RETURN;	                							
END_IF

	IF Execute
	THEN
		Error												:=	FALSE;
		ErrorId												:= 0;
		ItpResetEx2.bExecute 								:= rNCIRef.NciToPlc.ErrorCode <> 0;
	ELSIF NOT ItpSingleBlock.bBusy      					
	THEN                                					
		Error												:=	FALSE;
		ErrorId												:= 0;
		ItpResetEx2.bExecute 								:= FALSE;
	END_IF

	ItpResetEx2(
		bExecute	:= ,
		tTimeOut	:= ,
		sNciToPlc:= rNCIRef.NciToPlc,
		bBusy		=> Busy,
		bErr		=> ,
		nErrId	=> );

	Done													:= NOT ItpResetEx2.bBusy
																AND NOT ItpResetEx2.bErr
																AND ItpResetEx2.bExecute;

	IF NOT Busy
	THEN
		IF ItpResetEx2.bExecute
		THEN
			Error											:=	ItpResetEx2.bErr;
			ErrorId											:= ItpResetEx2.nErrId;
			ErrorText										:= SEL(Error , '' ,  CONCAT('Error ItpResetEx2 id: ',  UDINT_TO_STRING(Errorid)));
		END_IF                          					
		IF NOT Execute                  					
		THEN                            	
			MemFnc.4										:= FALSE ;
			ItpResetEx2(bExecute := FALSE, sNciToPlc:= rNCIRef.NciToPlc);
		END_IF
	END_IF
	
	reset													:= Busy;
END_METHOD

METHOD singleBlockModeChange : BOOL //Return = Busy
VAR_INPUT
	Execute													:	BOOL;
	SingleBlockMode											:	E_ItpSingleBlockMode;
END_VAR
IF NOT __ISVALIDREF(rNCIRef) 
THEN
	Busy													:= NOT Error;
	ErrorId													:= E_adsErr.DEVICE_INVALIDPARM;
	Error													:= TRUE;
	Done													:= FALSE;
	ErrorText												:= 'Reference to rNCIRef invalid (0)';
	RETURN;
END_IF
	
	IF Execute
	THEN
		Error												:=	FALSE;
		ErrorId												:= 0;
		ItpSingleBlock.bExecuteModeChange 					:= TRUE;
	ELSIF NOT ItpSingleBlock.bBusy	    					
	THEN                                					
		Error												:=	FALSE;
		ErrorId												:= 0;
		ItpSingleBlock.bExecuteModeChange 					:= FALSE;

	END_IF
	
	THIS^.SingleBlockMode									:= SingleBlockMode;
									
	ItpSingleBlock(
		bExecuteModeChange	:= ,
		nMode				:= SingleBlockMode,
		bTriggerNext		:=  ,
		tTimeOut			:= ,
		sNciToPlc			:= rNCIRef.NciToPlc,
		bBusy				=> Busy,
		bErr				=> ,
		nErrId				=> );

	Done													:= NOT ItpSingleBlock.bBusy
																AND NOT ItpSingleBlock.bErr
																AND ItpSingleBlock.bExecuteModeChange;

	IF NOT Busy
	THEN
		IF ItpSingleBlock.bExecuteModeChange
		THEN
			Error											:=	ItpSingleBlock.bErr;
			ErrorId											:= ItpSingleBlock.nErrId;
			ErrorText										:= CONCAT('Error ItpSingleBlock id: ',  UDINT_TO_STRING(Errorid));
		END_IF
		IF NOT Execute
		THEN
			MemFnc.5										:= FALSE;
			ItpSingleBlock(bExecuteModeChange := FALSE, sNciToPlc:= rNCIRef.NciToPlc);
		END_IF
	END_IF
	
	SingleBlockModeChange									:= Busy;
END_METHOD

METHOD PUBLIC singleBlockTrigNext : BOOL //Return value = TRUE if busy
//required parameter
//rNCIRef
VAR_INPUT
	Execute													:	BOOL;
END_VAR
IF NOT __ISVALIDREF(rNCIRef) 
THEN
	Busy													:= NOT Error;
	ErrorId													:= E_AdsErr.DEVICE_INVALIDPARM;
	Error													:= TRUE;
	Done													:= FALSE;
	ErrorText												:= 'Reference to rNCIRef invalid (0)';
	RETURN;
END_IF
	
	IF Execute
	THEN
		Error												:=	FALSE;
		ErrorId												:= 0;
		ItpSingleBlock.bTriggerNext 						:= TRUE ;
	ELSIF NOT ItpSingleBlock.bBusy	    					
	THEN                                					
		Error												:=	FALSE;
		ErrorId												:= 0;
		ItpSingleBlock.bTriggerNext 						:= FALSE;

	END_IF

	ItpSingleBlock(
		bExecuteModeChange	:= ,
		nMode				:= SingleBlockMode,
		bTriggerNext		:=  ,
		tTimeOut			:= ,
		sNciToPlc			:= rNCIRef.NciToPlc,
		bBusy				=> Busy,
		bErr				=> ,
		nErrId				=> );

	Done												:= NOT ItpSingleBlock.bBusy
															AND NOT ItpSingleBlock.bErr
															AND ItpSingleBlock.bTriggerNext;

	IF NOT Busy
	THEN
		IF ItpSingleBlock.bTriggerNext
		THEN
			Error										:=	ItpSingleBlock.bErr;
			ErrorId										:= ItpSingleBlock.nErrId;
			ErrorText									:= CONCAT('Error ItpSingleBlock id: ',  UDINT_TO_STRING(Errorid));
		END_IF
		IF NOT Execute
		THEN
			MemFnc.6									:= FALSE;
			ItpSingleBlock(bTriggerNext := FALSE, sNciToPlc:= rNCIRef.NciToPlc);
		END_IF
	END_IF
	
	SingleBlockTrigNext									:= Busy;
END_METHOD

END_FUNCTION_BLOCK

// POUs/Motion/TF5100-NCI/01_Main/NciGrp
{attribute 'no_check'}
//Nci group FB used to build,reconfig Nci groups as well to add and econfig single axis for group
//based on Tc2_NCI
FUNCTION_BLOCK NciGrp EXTENDS FbBase
VAR_OUTPUT CONSTANT
	FNC_BUILD												:	INT := 0; //Build Nci Grp
	FNC_RECONFIG											:	INT := 1; //Reconfig/loose group
	FNC_ADD_AXIS											:	INT := 2; //Add axis to group 
	FNC_RECONFIG_AXIS										:	INT := 3; //Reconfig axis out of grp
END_VAR                     								
VAR_INPUT                   								
	Fnc														:	INT (FNC_BUILD..FNC_RECONFIG_AXIS):= FNC_BUILD;
	XAxisId													: UDINT := 0;
	YAxisId													: UDINT := 0;
	ZAxisId													: UDINT := 0;
	Q1AxisId												: UDINT := 0;
	Q2AxisId												: UDINT := 0;
	Q3AxisId												: UDINT := 0;
	Q4AxisId												: UDINT := 0;
	Q5AxisId												: UDINT := 0;
	AxisIndex												:	NCI_AXCONFIG ;//contains the location of the axis within the group to add or release axis into group 
	rNCIRef													:	REFERENCE TO NCI_REF := 0;
END_VAR                         							
VAR_IN_OUT                      							
END_VAR                         							
VAR_OUTPUT                      							
	ErrorText												:	STRING(40);
END_VAR
VAR
(* Buffer **************************************************************************)
	MemFnc													:	INT := -1;

(* Trigger *)

(* Instanzierung der MC Bausteine *******************************************************)
	CfgBuildExt3DGroup										:	CfgBuildExt3DGroup := (tTimeOut	:= DEFAULT_ADS_TIMEOUT);
	CfgReconfigGroup										:	CfgReconfigGroup := (tTimeOut	:= DEFAULT_ADS_TIMEOUT);
	CfgReconfigAxis											:	CfgReconfigAxis := (tTimeOut	:= DEFAULT_ADS_TIMEOUT);
	CfgAddAxisToGroup										:	CfgAddAxisToGroup:= (tTimeOut	:= DEFAULT_ADS_TIMEOUT);

(* Dummy Speicher **********************************************************)
	K														:	UDINT;
END_VAR

	(* Nci Group control																*)
	(************************************************************************************)

(* Execute ***************************************************************************************)
	rtExecute(CLK := Execute );
	IF rtExecute.Q
		AND MemFnc < 0
	THEN
		MemFnc 												:= Fnc;
		Busy												:= TRUE;
		Done												:= FALSE;
		Error												:= FALSE;
		ErrorID												:= 0;
		ErrorText											:= '';
	END_IF

(* Call Method ***********************************************************************************)
	CASE MemFnc OF
	FNC_BUILD							:	
		Build(Execute	:= Execute);
			
	FNC_RECONFIG						:	
		Reconfig(Execute := Execute);
		
	FNC_ADD_AXIS						:
		CASE AxisIndex OF
		1:	K 												:= XAxisId;
		2:	K 												:= YAxisId;
		3:	K 												:= ZAxisId;
		4:	K 												:= Q1AxisId;
		5:	K 												:= Q2AxisId;
		6:	K 												:= Q3AxisId;
		7:	K 												:= Q4AxisId;
		8:	K 												:= Q5AxisId;
		ELSE
			K 												:= 0;
		END_CASE
		
		AddAxis(
			Execute		:= Execute,
			AxisIndex	:= AxisIndex,
			AxisId		:= k); //location of axis within a group

	FNC_RECONFIG_AXIS					:	

		CASE AxisIndex OF
		1 : K 												:= XAxisId;
		2:	K 												:= YAxisId;
		3:	K 												:= ZAxisId;
		4:	K 												:= Q1AxisId;
		5:	K 												:= Q2AxisId;
		6:	K 												:= Q3AxisId;
		7:	K 												:= Q4AxisId;
		8:	K 												:= Q5AxisId;
		ELSE
			K 												:= 0;
		END_CASE

		ReconfigAxis(
			Execute	:= Execute, 
			AxisId	:= K);
		
	-1:
		IF NOT Execute
		THEN
			Busy											:= FALSE;
			Done											:= FALSE;
			Error											:= FALSE;
			ErrorID											:= 0;
			ErrorText										:= '';
		END_IF                              				
	ELSE                                    				
		Busy												:= FALSE;
		Done												:= FALSE;
		Error												:= Execute;
		ErrorID												:= E_AdsErr.DEVICE_INVALIDPARM;
		ErrorText											:= CONCAT('invalid parameter value(s) Fnc no: ' , INT_TO_STRING(MemFnc));
	END_CASE


(**************************************************************************************************)

METHOD PUBLIC addAxis : BOOL //Return value = TRUE if busy
//required parameter
//rNCIRef
//AxisIndex -> XAxisId..Q5AxisId
VAR_INPUT
	Execute													:	BOOL;
	AxisIndex												:	NCI_AXCONFIG; //contains the location of the axis within the group
	AxisId													:	UDINT; //Axis ID which should be added to group - if 0 then ID of input parameters is used based on parameter AxisIndex
END_VAR
	MemFnc													:= FNC_ADD_AXIS;
	THIS^.Execute											:= Execute;
	THIS^.AxisIndex											:= AxisIndex;
	
IF NOT __ISVALIDREF(rNCIRef) 
THEN
	Busy													:= NOT Error;
	Error													:= TRUE;
	ErrorId													:= E_adsErr.DEVICE_INVALIDPARM;
	Done													:= FALSE;
	ErrorText												:= 'Reference to rNCIRef invalid (0)';
	MemFnc													:= SEL(Execute , -1 ,MemFnc);
	RETURN;
END_IF

	IF Execute
	THEN
		Error												:=	FALSE;
		ErrorId												:= 0;
		CfgAddAxisToGroup.bExecute 							:= TRUE;
	ELSIF NOT CfgAddAxisToGroup.bBusy   					
	THEN                                					
		Error												:=	FALSE;
		ErrorId												:= 0;
		CfgAddAxisToGroup.bExecute 							:= FALSE;

	END_IF
	
	IF AxisId > 0
	THEN
		CfgAddAxisToGroup.nAxisId							:= AxisId;
	ELSE		
		CASE AxisIndex OF
		1:	CfgAddAxisToGroup.nAxisId 						:= XAxisId ;
		2:	CfgAddAxisToGroup.nAxisId 						:= YAxisId ;
		3:	CfgAddAxisToGroup.nAxisId 						:= ZAxisId ;
		4:	CfgAddAxisToGroup.nAxisId 						:= Q1AxisId ;
		5:	CfgAddAxisToGroup.nAxisId 						:= Q2AxisId ;
		6:	CfgAddAxisToGroup.nAxisId 						:= Q3AxisId ;
		7:	CfgAddAxisToGroup.nAxisId 						:= Q4AxisId ;
		8:	CfgAddAxisToGroup.nAxisId 						:= Q5AxisId ;
		ELSE
			CfgAddAxisToGroup.nAxisId 						:= 0;
		END_CASE
	END_IF
	
	CfgAddAxisToGroup(
		bExecute	:= ,
		nGroupId	:= rNCIRef.NciToPlc.GrpId,
		nAxisId		:= ,
		nIndex		:= DINT_TO_UDINT(AxisIndex),
		tTimeOut	:= ,
		bBusy		=> busy,
		bErr		=> ,
		nErrId		=> );

	Done													:= NOT CfgAddAxisToGroup.bBusy
																AND NOT CfgAddAxisToGroup.bErr
																AND CfgAddAxisToGroup.bExecute;
                                        					
	IF NOT Busy                                         	
	THEN                                                	
		IF CfgAddAxisToGroup.bExecute                   	
		THEN                                            	
			Error											:=	CfgAddAxisToGroup.bErr;
			ErrorId											:= CfgAddAxisToGroup.nErrId;
			ErrorText										:= SEL(Error , '' ,  CONCAT('Error CfgAddAxisToGroup id: ',  UDINT_TO_STRING(Errorid)));
		END_IF                                          	
		IF NOT Execute                                  	
		THEN                                            	
			MemFnc											:= -1 ;
			CfgAddAxisToGroup(bExecute := FALSE);       	
		END_IF                                          	
	END_IF                                              	
                                                        	
	AddAxis													:= Busy;
END_METHOD

METHOD PUBLIC build : BOOL //Return value = TRUE if busy
//required parameter
//rNCIRef
//XAxisId
//YAxisId
//ZAxisId
//Q1AxisId
//Q2AxisId
//Q3AxisId
//Q4AxisId
//Q5AxisId
VAR_INPUT
	Execute													:	BOOL;
END_VAR
	MemFnc													:= FNC_BUILD;
	THIS^.Execute											:= Execute;
	
IF NOT __ISVALIDREF(rNCIRef) 
THEN
	Busy													:= NOT Error;
	Error													:= TRUE;
	ErrorId													:= E_AdsErr.DEVICE_INVALIDPARM;
	Done													:= FALSE;
	ErrorText												:= 'Reference to rNCIRef invalid (0)';
	MemFnc													:= SEL(Execute , -1 ,MemFnc);
	RETURN;                                             	
END_IF

	IF Execute
	THEN
		Error												:=	FALSE;
		ErrorId												:= 0;
		CfgBuildExt3DGroup.bExecute 						:= TRUE;
	ELSIF NOT CfgBuildExt3DGroup.bBusy  					
	THEN                                					
		Error												:=	FALSE;
		ErrorId												:= 0;
		CfgBuildExt3DGroup.bExecute 						:= FALSE;
                                        	
	END_IF

	CfgBuildExt3DGroup(
		bExecute	:= ,
		nGroupId	:= rNciRef.NciToPlc.GrpId,
		nXAxisId	:= XAxisId,
		nYAxisId	:= YAxisId,
		nZAxisId	:= ZAxisId,
		nQ1AxisId	:= Q1AxisId,
		nQ2AxisId	:= Q2AxisId,
		nQ3AxisId	:= Q3AxisId,
		nQ4AxisId	:= Q4AxisId,
		nQ5AxisId	:= Q5AxisId,
		tTimeOut	:= ,
		bBusy		=> busy,
		bErr		=> ,
		nErrId	=> );

	Done													:= NOT CfgBuildExt3DGroup.bBusy
																AND NOT CfgBuildExt3DGroup.bErr
																AND CfgBuildExt3DGroup.bExecute;
                                        					
	IF NOT Busy
	THEN
		IF CfgBuildExt3DGroup.bExecute
		THEN
			Error											:=	CfgBuildExt3DGroup.bErr;
			ErrorId											:= CfgBuildExt3DGroup.nErrId;
			ErrorText										:= SEL(Error , '' ,  CONCAT('Error CfgBuildExt3DGroup id: ',  UDINT_TO_STRING(Errorid)));
		END_IF
		IF NOT Execute
		THEN
			MemFnc											:= -1 ;
			CfgBuildExt3DGroup(bExecute := FALSE);
		END_IF
	END_IF

	Build													:= Busy;
END_METHOD

METHOD PUBLIC reconfig : BOOL //Return value = TRUE if busy
//required parameter
//rNCIRef
VAR_INPUT
	Execute													:	BOOL;
END_VAR

	MemFnc													:= FNC_RECONFIG;
	THIS^.Execute											:= Execute;
	
IF NOT __ISVALIDREF(rNCIRef) THEN
	Busy													:= NOT Error;
	Error													:= TRUE;
	ErrorId													:= E_AdsErr.DEVICE_INVALIDPARM;
	Done													:= FALSE;
	ErrorText												:= 'Reference to rNCIRef invalid (0)';
	MemFnc													:= SEL(Execute , -1 ,MemFnc);
	RETURN;
END_IF

	IF Execute
	THEN
		Error												:=	FALSE;
		ErrorId												:= 0;
		CfgReconfigGroup.bExecute 							:= TRUE;
	ELSIF NOT CfgReconfigGroup.bBusy    					
	THEN                                					
		Error												:=	FALSE;
		ErrorId												:= 0;
		CfgReconfigGroup.bExecute 							:= FALSE;

	END_IF

	CfgReconfigGroup(
		bExecute	:= ,
		nGroupId	:= rNCIRef.NciToPlc.GrpId,
		tTimeOut	:= ,
		bBusy		=> busy,
		bErr		=> ,
		nErrId		=> );

	Done													:= NOT CfgReconfigGroup.bBusy
																AND NOT CfgReconfigGroup.bErr
																AND CfgReconfigGroup.bExecute;
                                        					
	IF NOT Busy
	THEN
		IF CfgReconfigGroup.bExecute
		THEN
			Error											:=	CfgReconfigGroup.bErr;
			ErrorId											:= CfgReconfigGroup.nErrId;
			ErrorText										:= SEL(Error , '' ,  CONCAT('Error CfgReconfigGroup id: ',  UDINT_TO_STRING(Errorid)));
		END_IF                      						
		IF NOT Execute              						
		THEN                        						
			MemFnc											:= -1 ;
			CfgReconfigGroup(bExecute := FALSE,);
		END_IF
	END_IF
	
	Reconfig												:= Busy;
END_METHOD

METHOD PUBLIC reconfigAxis : BOOL //Return value = TRUE if busy
//required parameter
//rNCIRef
//AxisId
VAR_INPUT
	Execute													:	BOOL;
	AxisId													:	UDINT; //Axis ID which should be released from group - if 0 then ID of input parameters is used based on parameter AxisIndex
END_VAR
	MemFnc													:= FNC_ADD_AXIS;
	THIS^.Execute											:= Execute;
	
IF NOT __ISVALIDREF(rNCIRef) THEN
	Busy													:= NOT Error;
	Error													:= TRUE;
	ErrorId													:= E_AdsErr.DEVICE_INVALIDPARM;
	Done													:= FALSE;
	ErrorText												:= 'Reference to rNCIRef invalid (0)';
	MemFnc													:= SEL(Execute , -1 ,MemFnc);
	RETURN;
END_IF

	IF Execute
	THEN
		Error												:=	FALSE;
		ErrorId												:= 0;
		CfgReconfigAxis.bExecute 							:= TRUE;
	ELSIF NOT CfgReconfigAxis.bBusy     					
	THEN                                					
		Error												:=	FALSE;
		ErrorId												:= 0;
		CfgReconfigAxis.bExecute 							:= FALSE;

	END_IF

	IF AxisId > 0
	THEN
		CfgReconfigAxis.nAxisId								:= AxisId;
	ELSE
		CASE AxisIndex OF
		1:	CfgReconfigAxis.nAxisId 						:= XAxisId ;
		2:	CfgReconfigAxis.nAxisId 						:= YAxisId ;
		3:	CfgReconfigAxis.nAxisId 						:= ZAxisId ;
		4:	CfgReconfigAxis.nAxisId 						:= Q1AxisId ;
		5:	CfgReconfigAxis.nAxisId 						:= Q2AxisId ;
		6:	CfgReconfigAxis.nAxisId 						:= Q3AxisId ;
		7:	CfgReconfigAxis.nAxisId 						:= Q4AxisId ;
		8:	CfgReconfigAxis.nAxisId 						:= Q5AxisId ;
		ELSE
			CfgReconfigAxis.nAxisId 						:= 0;
		END_CASE
	END_IF

	CfgReconfigAxis(
		bExecute	:= ,
		nAxisId		:= ,
		tTimeOut	:= ,
		bBusy		=> busy,
		bErr		=> ,
		nErrId		=> );

	Done													:= NOT CfgReconfigAxis.bBusy
																AND NOT CfgReconfigAxis.bErr
																AND CfgReconfigAxis.bExecute;
                                        					
	IF NOT Busy
	THEN
		IF CfgReconfigAxis.bExecute
		THEN
			Error											:=	CfgReconfigAxis.bErr;
			ErrorId											:= CfgReconfigAxis.nErrId;
			ErrorText										:= SEL(Error , '' ,  CONCAT('Error CfgReconfigAxis id: ',  UDINT_TO_STRING(Errorid)));
		END_IF
		IF NOT Execute
		THEN
			MemFnc											:= -1 ;
			CfgReconfigAxis(bExecute := FALSE);
		END_IF
	END_IF
	
	ReconfigAxis											:= Busy;
END_METHOD

END_FUNCTION_BLOCK

// POUs/Motion/TF5100-NCI/01_Main/NciItp
//Nci Interpolation group control - load,start,stop Nci programs as well start interpolated moves via Plc table (Tc2_PlcInterpolation library)
//based on Tc2_NCI, TcNcCfg.lib, Tc2_PlcInterpolation librarys
FUNCTION_BLOCK NciItp  EXTENDS FbBase
VAR_OUTPUT CONSTANT
	FNC_RESET												:	INT := 0; //Reset Nci group
	FNC_LOAD												:	INT := 1; //Load Nci program as txt/nc file
	FNC_START												:	INT := 2; //Start loaded Nci program
	FNC_STOP												:	INT := 3; //Stop loaded Nci programm
	FNC_FEED_TBL											:	INT := 4; //Feed table group - provided by Tc2_PlcInterpolation library
END_VAR                     								
VAR_INPUT                   								
	Fnc														:	INT (FNC_RESET..FNC_FEED_TBL):= FNC_RESET;
	Prg														:	T_MaxString := '';	//Program
	rTable													:	REFERENCE TO ST_NciFeedGroupTable := 0; //-> NciItpTableEntry
	rNCIRef													:	REFERENCE TO NCI_REF := 0;
	StartPrgAfterLoading									:	BOOL := FALSE; //Return value TRUE = Start Program direct after loading 
	LogFeederEntries										:	BOOL := FALSE; //Return value TRUE = Log tabel entries by Fnc FeedTbl
	WaitForChnDoneByEndOfTbl								:	BOOL := FALSE; //Fnc FeedTabl - TRUE = FB is busy as long as the prg is running if table contains entry "ST_NciEndOfTables"
END_VAR                     								
VAR_IN_OUT                  								
END_VAR                     								
VAR_OUTPUT                  								
	ErrorText												:	STRING(40);
END_VAR
VAR
(* cache **************************************************************************)
	MemFnc													:	INT := -1;
	MemResetAfterStop										:	BOOL;
                            								
(* timer *)                 								
                            	
(* trigger *)               	

(* MC-Function-block intances ******************************************************)
	ItpLoadProgEx											:	ItpLoadProgEx;
	ItpStartStopEx											:	ItpStartStopEx;
	NciFeedTable											:	FB_NciFeedTable;
	ItpResetEx2												:	ItpResetEx2 := (tTimeOut	:= DEFAULT_ADS_TIMEOUT);

END_VAR

	(* NCI Program control																*)
	(************************************************************************************)

(* Execute ***************************************************************************************)
	rtExecute(CLK := Execute );
	IF rtExecute.Q
		AND MemFnc < 0
	THEN
		MemFnc 												:= Fnc;
		Busy												:= TRUE;
		Done												:= FALSE;
		Error												:= FALSE;
		ErrorID												:= 0;
		ErrorText											:= '';
	END_IF

(* Call Method ***********************************************************************************)
	CASE MemFnc OF
	FNC_RESET							:
		Reset(Execute:= Execute);
	FNC_LOAD							:
		LoadPrg(Execute:= Execute, Prg:= Prg);
	FNC_START							:
		StartPrg(Execute:= Execute);
	FNC_STOP							:
		StopPrg(Execute:= Execute);
	FNC_FEED_TBL						:
		FeedTbl(Execute:= Execute );
	-1:
		IF NOT Execute
		THEN
			Busy											:= FALSE;
			Done											:= FALSE;
			Error											:= FALSE;
			ErrorID											:= 0;
			ErrorText										:= '';
		END_IF                              				
	ELSE                                    				
		Busy												:= FALSE;
		Done												:= FALSE;
		Error												:= Execute;
		ErrorID												:= E_AdsErr.DEVICE_INVALIDPARM;
		ErrorText											:= CONCAT('invalid parameter value(s) Fnc no: ' , INT_TO_STRING(MemFnc));
	END_CASE


(**************************************************************************************************)

METHOD PUBLIC feedTbl : BOOL //Return value = TRUE if busy
//required parameter
//rNCIRef
//rTable
VAR_INPUT
	Execute													:	BOOL := FALSE;
END_VAR
	MemFnc													:= FNC_FEED_TBL;
	THIS^.Execute											:= Execute;
	
IF NOT __ISVALIDREF(rNCIRef) 
THEN
	Busy													:= NOT Error;
	Error													:= TRUE;
	ErrorId													:= E_AdsErr.DEVICE_INVALIDPARM;
	Done													:= FALSE;
	ErrorText												:= 'Reference rNCIRef invalid (0)';
	MemFnc													:= SEL(Execute , -1 ,MemFnc); 
	RETURN;
ELSIF NOT __ISVALIDREF(rTable) 
THEN
	Busy													:= NOT Error;
	Error													:= TRUE;
	ErrorId													:= E_AdsErr.DEVICE_INVALIDPARM;
	Done													:= FALSE;
	ErrorText												:= 'Reference rTable invalid (0)';
	MemFnc													:= SEL(Execute , -1 ,MemFnc);
	RETURN;
END_IF

	IF Execute
	THEN
		Error												:=	FALSE;
		ErrorId												:= 0;
		NciFeedTable.bExecute 								:= TRUE;
	ELSIF NOT NciFeedTable.bFeedBusy
		AND(
		NOT NciFeedTable.bExecChannelDoneCheck
		OR NciFeedTable.bChannelDone)
	THEN
		Error												:=	FALSE;
		ErrorId												:= 0;
		NciFeedTable.bExecute 								:= FALSE;
	END_IF

	NciFeedTable(
		bExecute			:= ,
		bReset				:= FALSE,
		bLogFeederEntries	:= LogFeederEntries,
		stFeedGroupTable	:= rTable,
		stNciToPlc			:= rNCIRef.NciToPlc,
		bFeedingDone		=> 	,
		bChannelDone		=> ,
		bFeedBusy			=> ,
		bResetBusy			=> ,
		bError				=> ,
		nErrorId			=> );

	IF WaitForChnDoneByEndOfTbl
	THEN
		Busy 												:= NciFeedTable.bFeedBusy
																OR
																NciFeedTable.bFeedingDone
																AND NciFeedTable.bExecChannelDoneCheck
																AND NOT NciFeedTable.bChannelDone;
                            								
		Done												:= NciFeedTable.bChannelDone
																OR
																NciFeedTable.bFeedingDone
																AND NOT NciFeedTable.bExecChannelDoneCheck;
                            								
	ELSE                    								
		Busy												:= NciFeedTable.bFeedBusy;
		Done												:= NciFeedTable.bFeedingDone;
	END_IF

	IF NOT Busy
	THEN
		IF NciFeedTable.bExecute
		THEN
			Error											:=	NciFeedTable.bError;
			ErrorId											:= NciFeedTable.nErrorId;
			ErrorText										:= SEL(Error , '' ,  CONCAT('Error NciFeedTable id: ',  UDINT_TO_STRING(Errorid)));
		END_IF                          					
		IF NOT Execute                  					
		THEN                            					
			MemFnc											:= -1 ;
			NciFeedTable(bExecute 							:= FALSE, stNciToPlc:= rNCIRef.NciToPlc, stFeedGroupTable:= rTable  );
		END_IF                          	
	END_IF                              	
                                        	
	FeedTbl													:= Busy;
END_METHOD

METHOD PUBLIC loadPrg : BOOL //Return value = TRUE if busy
//required parameter
//rNCIRef
VAR_INPUT
	Execute													:	BOOL;
	Prg														:	T_MaxString := ''; //if Prg = '' then INPUT THIS^.Prg used
END_VAR
	MemFnc													:= FNC_LOAD;
	THIS^.Execute											:= Execute;
	
IF NOT __ISVALIDREF(rNCIRef) THEN
	Busy													:= NOT Error;
	Error													:= TRUE;
	ErrorId													:= E_AdsErr.DEVICE_INVALIDPARM;
	Done													:= FALSE;
	ErrorText												:= 'Reference rNCIRef invalid (0)';
	MemFnc													:= SEL(Execute , -1 ,MemFnc);
	RETURN;
END_IF
	
	IF Execute AND NOT ItpLoadProgEx.bExecute
	THEN
		IF LEN(Prg) > 0
		THEN
			ItpLoadProgEx.sPrg								:= Prg;
		ELSE                    							
			ItpLoadProgEx.sPrg								:= THIS^.Prg;	
		END_IF
	END_IF	
	
	IF Execute
	THEN
		Error												:=	FALSE;
		ErrorId												:= 0;
		ItpLoadProgEx.bExecute 								:= TRUE;
	ELSIF NOT ItpLoadProgEx.bBusy       					
		AND(                            					
		NOT ItpStartStopEx.bBusy        					
		OR NOT StartPrgAfterLoading)    					
	THEN                                					
		Error												:=	FALSE;
		ErrorId												:= 0;
		ItpLoadProgEx.bExecute 								:= FALSE;
		IF StartPrgAfterLoading             				
		THEN                                				
			ItpStartStopEx.bStart 							:= FALSE;
		END_IF
	END_IF
	
	ItpLoadProgEx(
		bExecute	:= ,
		sPrg		:= ,
		nLength		:= INT_TO_UDINT(LEN(Prg)),
		tTimeOut	:= ,
		sNciToPlc	:= rNCIRef.NciToPlc,
		bBusy		=> ,
		bErr		=> ,
		nErrId		=> );

	IF StartPrgAfterLoading
		OR ItpStartStopEx.bBusy
	THEN
		ItpStartStopEx(
			bStart		:= ItpLoadProgEx.bExecute
							AND NOT ItpLoadProgEx.bErr
							AND NOT ItpLoadProgEx.bBusy,
			bStop		:= FALSE,
			tTimeOut	:=  ,
			sNciToPlc	:= rNCIRef.NciToPlc,
			bBusy		=> ,
			bErr		=> ,
			nErrId		=> );
	END_IF


	Busy													:= ItpStartStopEx.bBusy OR ItpLoadProgEx.bBusy;
                                        					
	IF StartPrgAfterLoading             					
	THEN                                					
		Done												:= NOT Busy
																AND NOT ItpStartStopEx.bErr
																AND ItpStartStopEx.bStart;
	ELSE                                	    		
		Done												:= NOT Busy
																AND NOT ItpLoadProgEx.bErr
																AND ItpLoadProgEx.bExecute;
	END_IF                                      		
                                                	
	IF NOT Busy                                 	
	THEN
		IF ItpLoadProgEx.bExecute
			AND NOT StartPrgAfterLoading
		THEN
			Error											:=	ItpLoadProgEx.bErr;
			ErrorId											:= ItpLoadProgEx.nErrId;
			ErrorText										:= SEL(Error , '' ,  CONCAT('Error ItpLoadProgEx id: ',  UDINT_TO_STRING(Errorid)));
		ELSIF ItpStartStopEx.bStart 						
		THEN                        						
			Error												:=	ItpStartStopEx.bErr;
			ErrorId											:= ItpStartStopEx.nErrId;
			ErrorText										:= SEL(Error , '' ,  CONCAT('Error ItpStartStopEx id: ',  UDINT_TO_STRING(Errorid)));
		END_IF                          					
                                        					
		IF NOT Execute                  	
		THEN                            	
			MemFnc											:= -1 ;
			ItpLoadProgEx(bExecute := FALSE, sNciToPlc:= rNCIRef.NciToPlc);
			IF StartPrgAfterLoading
			THEN
				ItpStartStopEx(bStart := FALSE, sNciToPlc:= rNCIRef.NciToPlc);
			END_IF
		END_IF
	END_IF
	
	LoadPrg													:= Busy;
END_METHOD

METHOD PUBLIC reset : BOOL //Return value = TRUE if busy
//required parameter
//rNCIRef
//rTable
VAR_INPUT	
	Execute													:	BOOL := FALSE;
END_VAR
	MemFnc													:= FNC_RESET;
	THIS^.Execute											:= Execute;
	
IF NOT __ISVALIDREF(rNCIRef) 
THEN
	Busy													:= NOT Error;
	Error													:= TRUE;
	ErrorId													:= E_AdsErr.DEVICE_INVALIDPARM;
	Done													:= FALSE;
	ErrorText												:= 'Reference rNCIRef invalid (0)';
	MemFnc													:= SEL(Execute , -1 ,MemFnc);
	RETURN;
ELSIF NOT __ISVALIDREF(rTable) AND FALSE 
THEN
	Busy													:= NOT Error;
	Error													:= TRUE;
	ErrorId													:= E_AdsErr.DEVICE_INVALIDPARM;
	Done													:= FALSE;
	ErrorText												:= 'Reference rTable invalid (0)';
	MemFnc													:= SEL(Execute , -1 ,MemFnc);
	RETURN;
END_IF

IF Execute
THEN
	Error													:=	FALSE;
	ErrorId													:= 0;
	NciFeedTable.bReset 									:= __ISVALIDREF(rTable);
	ItpResetEx2.bExecute									:= NOT __ISVALIDREF(rTable);
ELSIF NOT NciFeedTable.bFeedBusy                        	
AND NOT ItpResetEx2.bBusy                               	
THEN                                                    	
	Error													:=	FALSE;
	ErrorId													:= 0;
	NciFeedTable.bReset 									:= FALSE;
	ItpResetEx2.bExecute									:= FALSE; 
END_IF

IF	NOT __ISVALIDREF(rTable)
THEN
	ItpResetEx2(
		bExecute	:= ,
		tTimeOut	:= ,
		sNciToPlc	:= rNCIRef.NciToPlc,
		bBusy		=> Busy,
		bErr		=> ,
		nErrId		=> );
ELSE
	NciFeedTable(
		bExecute			:= FALSE,
		bReset				:= ,
		bLogFeederEntries	:= ,
		stFeedGroupTable	:= rTable,
		stNciToPlc			:= rNCIRef.NciToPlc,
		bFeedingDone		=> ,
		bChannelDone		=> ,
		bFeedBusy			=> ,
		bResetBusy			=> busy,
		bError				=> ,
		nErrorId			=> );
END_IF
Done														:= NOT NciFeedTable.bResetBusy AND NOT ItpResetEx2.bBusy
															 	AND NOT NciFeedTable.bError AND NOT ItpResetEx2.bErr
															 	AND(NciFeedTable.bReset OR ItpResetEx2.bExecute);
                                                      	     
